KUKA KRL program: MyProgram_135().src

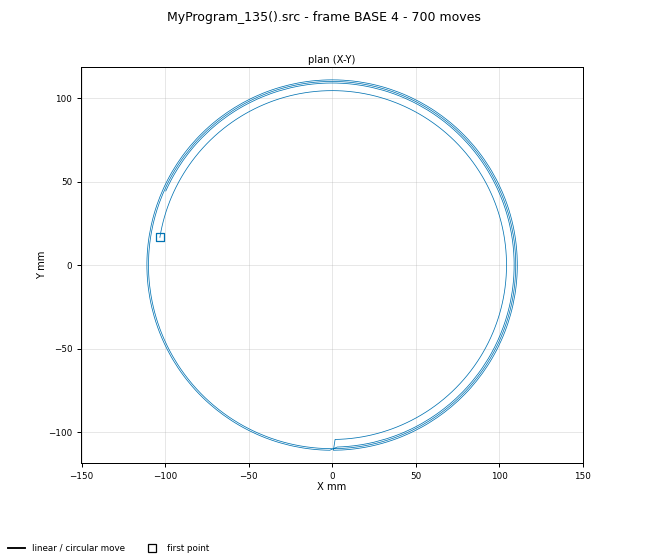
[picture p0: tool path of MyProgram_135().src in frame BASE 4, 700 of 700 moves have a stored position in this frame; points joined in program order, loops and branches not executed]
&ACCESS RVP
&REL 1
&PARAM TEMPLATE = C:\KRC\Roboter\Template\vorgabe
&PARAM EDITMASK = *
DEF MyProgram_135()
; ---- Setting reference (Base) ----
$BASE = BASE_DATA[4]

; --------------------------
; ---- Setting tool (TCP) ----
$TOOL = TOOL_DATA[3]
; --------------------------

$VEL.CP = VEL_APROX_PRINT
Startdeposition()
$VEL.CP = VEL_PRINT
LIN {X -103.1333,Y 16.5825,Z 109,A 165.9038,B 24.9354,C -1.8568,E1 24.8421,E2 279.7377} C_DIS
LIN {X -102.5383,Y 19.9247,Z 109,A 164.1624,B 24.9347,C -1.867,E1 24.843,E2 281.465} C_DIS
LIN {X -101.9199,Y 22.8869,Z 109,A 162.3578,B 24.9347,C -1.8672,E1 24.844,E2 283.2797} C_DIS
LIN {X -101.1577,Y 26.042,Z 109,A 160.77,B 24.9338,C -1.8797,E1 24.8451,E2 284.8471} C_DIS
LIN {X -100.4534,Y 28.6392,Z 109,A 159.199,B 24.9337,C -1.881,E1 24.8463,E2 286.424} C_DIS
LIN {X -99.4092,Y 32.0762,Z 109,A 157.2856,B 24.9331,C -1.8892,E1 24.8479,E2 288.3288} C_DIS
LIN {X -98.5325,Y 34.676,Z 109,A 155.6889,B 24.933,C -1.8907,E1 24.8493,E2 289.9311} C_DIS
LIN {X -97.2525,Y 38.1187,Z 109,A 153.7477,B 24.9324,C -1.8995,E1 24.8512,E2 291.8622} C_DIS
LIN {X -96.2896,Y 40.4893,Z 109,A 152.276,B 24.9322,C -1.9014,E1 24.8528,E2 293.3376} C_DIS
LIN {X -94.9474,Y 43.5478,Z 109,A 150.3049,B 24.9322,C -1.902,E1 24.8551,E2 295.318} C_DIS
LIN {X -93.5406,Y 46.4891,Z 109,A 148.6045,B 24.9316,C -1.9105,E1 24.8571,E2 297.0073} C_DIS
LIN {X -91.8565,Y 49.7339,Z 109,A 146.632,B 24.9311,C -1.9176,E1 24.8597,E2 298.9735} C_DIS
LIN {X -90.2584,Y 52.582,Z 109,A 144.8687,B 24.9306,C -1.9237,E1 24.8621,E2 300.7314} C_DIS
LIN {X -88.786,Y 55.0296,Z 109,A 143.2,B 24.9306,C -1.9246,E1 24.8646,E2 302.4065} C_DIS
LIN {X -87.1648,Y 57.5619,Z 109,A 141.5447,B 24.9302,C -1.9291,E1 24.8671,E2 304.0595} C_DIS
LIN {X -85.388,Y 60.1693,Z 109,A 139.8581,B 24.9298,C -1.9354,E1 24.8698,E2 305.7393} C_DIS
LIN {X -83.8937,Y 62.2359,Z 109,A 138.3455,B 24.9298,C -1.9352,E1 24.8723,E2 307.2598} C_DIS
LIN {X -81.9529,Y 64.7672,Z 109,A 136.6672,B 24.9293,C -1.9424,E1 24.8751,E2 308.9288} C_DIS
LIN {X -79.7445,Y 67.4686,Z 109,A 134.6792,B 24.9291,C -1.9448,E1 24.8787,E2 310.9204} C_DIS
LIN {X -77.5632,Y 69.9655,Z 109,A 132.8296,B 24.9288,C -1.9483,E1 24.8821,E2 312.7698} C_DIS
LIN {X -75.2059,Y 72.4924,Z 109,A 130.9953,B 24.9283,C -1.9552,E1 24.8856,E2 314.5956} C_DIS
LIN {X -72.7466,Y 74.9609,Z 109,A 129.0328,B 24.9281,C -1.9579,E1 24.8895,E2 316.5599} C_DIS
LIN {X -70.3326,Y 77.2305,Z 109,A 127.1463,B 24.928,C -1.9597,E1 24.8934,E2 318.4498} C_DIS
LIN {X -67.7352,Y 79.5174,Z 109,A 125.3395,B 24.9274,C -1.9673,E1 24.8972,E2 320.2456} C_DIS
LIN {X -64.9962,Y 81.7719,Z 109,A 123.3659,B 24.9272,C -1.9706,E1 24.9015,E2 322.2189} C_DIS
LIN {X -62.8029,Y 83.4678,Z 109,A 121.8583,B 24.9269,C -1.9743,E1 24.9048,E2 323.7231} C_DIS
LIN {X -60.123,Y 85.4206,Z 109,A 119.9594,B 24.9269,C -1.975,E1 24.9091,E2 325.6268} C_DIS
LIN {X -57.3874,Y 87.2798,Z 109,A 118.158,B 24.9266,C -1.9791,E1 24.9133,E2 327.4244} C_DIS
LIN {X -54.2739,Y 89.2491,Z 109,A 116.2553,B 24.926,C -1.9872,E1 24.9178,E2 329.314} C_DIS
LIN {X -52.1167,Y 90.5258,Z 109,A 114.8585,B 24.9258,C -1.9889,E1 24.9211,E2 330.7109} C_DIS
LIN {X -49.7124,Y 91.8681,Z 109,A 113.2634,B 24.9258,C -1.9884,E1 24.9251,E2 332.3118} C_DIS
LIN {X -46.4551,Y 93.5574,Z 109,A 111.2906,B 24.9255,C -1.9931,E1 24.93,E2 334.2786} C_DIS
LIN {X -43.4974,Y 94.9708,Z 109,A 109.3318,B 24.9257,C -1.99,E1 24.9349,E2 336.2497} C_DIS
LIN {X -40.495,Y 96.2872,Z 109,A 107.6366,B 24.9253,C -1.9964,E1 24.9393,E2 337.9336} C_DIS
LIN {X -37.0875,Y 97.6504,Z 109,A 105.6975,B 24.9249,C -2.0019,E1 24.9443,E2 339.8639} C_DIS
LIN {X -34.6623,Y 98.5373,Z 109,A 104.2027,B 24.9249,C -2.0008,E1 24.9482,E2 341.3642} C_DIS
LIN {X -31.5292,Y 99.586,Z 109,A 102.2735,B 24.9251,C -1.9986,E1 24.9534,E2 343.3022} C_DIS
LIN {X -28.5461,Y 100.4798,Z 109,A 100.7134,B 24.9246,C -2.006,E1 24.9575,E2 344.8473} C_DIS
LIN {X -25.3785,Y 101.3282,Z 109,A 98.7564,B 24.9249,C -2.0018,E1 24.9628,E2 346.817} C_DIS
LIN {X -22.3293,Y 102.0416,Z 109,A 97.2308,B 24.9242,C -2.0106,E1 24.9669,E2 348.3238} C_DIS
LIN {X -19.631,Y 102.5949,Z 109,A 95.6315,B 24.9244,C -2.0085,E1 24.9713,E2 349.9298} C_DIS
LIN {X -16.2066,Y 103.1915,Z 109,A 93.7524,B 24.9242,C -2.0109,E1 24.9765,E2 351.8049} C_DIS
LIN {X -13.3362,Y 103.6013,Z 109,A 92.1299,B 24.9242,C -2.0107,E1 24.981,E2 353.4292} C_DIS
LIN {X -9.5889,Y 104.015,Z 109,A 90.1169,B 24.924,C -2.0139,E1 24.9866,E2 355.4358} C_DIS
LIN {X -6.3744,Y 104.2632,Z 109,A 88.1851,B 24.9244,C -2.0084,E1 24.992,E2 357.3813} C_DIS
LIN {X -3.091,Y 104.4104,Z 109,A 86.4916,B 24.924,C -2.0132,E1 24.9967,E2 359.0639} C_DIS
LIN {X 0.6428,Y 104.4541,Z 109,A 84.5244,B 24.9237,C -2.0167,E1 25.0022,E2 361.0227} C_DIS
LIN {X 3.337,Y 104.4028,Z 109,A 82.9539,B 24.924,C -2.0133,E1 25.0066,E2 362.6009} C_DIS
LIN {X 6.4284,Y 104.2599,Z 109,A 81.1548,B 24.9243,C -2.0094,E1 25.0116,E2 364.4086} C_DIS
LIN {X 9.683,Y 104.0063,Z 109,A 79.4608,B 24.924,C -2.013,E1 25.0163,E2 366.0931} C_DIS
LIN {X 13.3502,Y 103.5994,Z 109,A 77.4906,B 24.9239,C -2.0147,E1 25.0217,E2 368.0578} C_DIS
LIN {X 16.6067,Y 103.1294,Z 109,A 75.5342,B 24.9244,C -2.0083,E1 25.0272,E2 370.0277} C_DIS
LIN {X 19.6735,Y 102.5867,Z 109,A 73.9793,B 24.924,C -2.0136,E1 25.0314,E2 371.5683} C_DIS
LIN {X 22.8843,Y 101.9205,Z 109,A 72.0241,B 24.9245,C -2.0066,E1 25.0368,E2 373.5375} C_DIS
LIN {X 25.9326,Y 101.1858,Z 109,A 70.5056,B 24.924,C -2.0134,E1 25.0408,E2 375.0374} C_DIS
LIN {X 28.5921,Y 100.4668,Z 109,A 68.9194,B 24.9243,C -2.0095,E1 25.0451,E2 376.6305} C_DIS
LIN {X 32.0776,Y 99.4088,Z 109,A 66.9893,B 24.9243,C -2.0106,E1 25.0503,E2 378.5544} C_DIS
LIN {X 34.6913,Y 98.5271,Z 109,A 65.4074,B 24.9245,C -2.0066,E1 25.0545,E2 380.1427} C_DIS
LIN {X 38.1127,Y 97.2548,Z 109,A 63.4873,B 24.9245,C -2.0079,E1 25.0595,E2 382.0555} C_DIS
LIN {X 40.5037,Y 96.2836,Z 109,A 62.0408,B 24.9246,C -2.0052,E1 25.0632,E2 383.5051} C_DIS
LIN {X 43.5071,Y 94.9663,Z 109,A 60.0932,B 24.9252,C -1.9972,E1 25.0682,E2 385.4667} C_DIS
LIN {X 46.4667,Y 93.5517,Z 109,A 58.4072,B 24.925,C -1.9995,E1 25.0724,E2 387.1429} C_DIS
LIN {X 49.7271,Y 91.8602,Z 109,A 56.4415,B 24.925,C -1.9988,E1 25.0772,E2 389.1048} C_DIS
LIN {X 52.602,Y 90.2469,Z 109,A 54.6726,B 24.9252,C -1.9977,E1 25.0815,E2 390.8709} C_DIS
LIN {X 54.8087,Y 88.9239,Z 109,A 53.0827,B 24.9259,C -1.9884,E1 25.0854,E2 392.4777} C_DIS
LIN {X 57.567,Y 87.1614,Z 109,A 51.3965,B 24.9257,C -1.99,E1 25.0893,E2 394.1548} C_DIS
LIN {X 60.5312,Y 85.1297,Z 109,A 49.4373,B 24.926,C -1.9871,E1 25.0938,E2 396.1139} C_DIS
LIN {X 63.2881,Y 83.1026,Z 109,A 47.5197,B 24.9263,C -1.9821,E1 25.0981,E2 398.0364} C_DIS
LIN {X 65.78,Y 81.1422,Z 109,A 45.8503,B 24.9263,C -1.9818,E1 25.1017,E2 399.7005} C_DIS
LIN {X 68.4304,Y 78.9208,Z 109,A 43.9194,B 24.9267,C -1.9767,E1 25.1058,E2 401.6359} C_DIS
LIN {X 70.8883,Y 76.7206,Z 109,A 42.0884,B 24.9271,C -1.9721,E1 25.1096,E2 403.4702} C_DIS
LIN {X 73.4416,Y 74.2792,Z 109,A 40.2308,B 24.9271,C -1.9713,E1 25.1133,E2 405.322} C_DIS
LIN {X 75.8718,Y 71.7958,Z 109,A 38.2991,B 24.9275,C -1.9661,E1 25.1171,E2 407.2577} C_DIS
LIN {X 78.0198,Y 69.4555,Z 109,A 36.5169,B 24.9279,C -1.9605,E1 25.1204,E2 409.0452} C_DIS
LIN {X 80.342,Y 66.7551,Z 109,A 34.6539,B 24.9279,C -1.9597,E1 25.1238,E2 410.9017} C_DIS
LIN {X 82.571,Y 63.978,Z 109,A 32.7197,B 24.9283,C -1.9557,E1 25.1271,E2 412.8361} C_DIS
LIN {X 84.3727,Y 61.5819,Z 109,A 31.0746,B 24.9286,C -1.9516,E1 25.1299,E2 414.483} C_DIS
LIN {X 86.1363,Y 59.0932,Z 109,A 29.2885,B 24.9292,C -1.9427,E1 25.1327,E2 416.2815} C_DIS
LIN {X 87.944,Y 56.3643,Z 109,A 27.6077,B 24.9292,C -1.9427,E1 25.1353,E2 417.9536} C_DIS
LIN {X 89.8865,Y 53.2117,Z 109,A 25.6766,B 24.9293,C -1.9415,E1 25.1381,E2 419.8778} C_DIS
LIN {X 91.1627,Y 50.9945,Z 109,A 24.2402,B 24.9297,C -1.9364,E1 25.14,E2 421.319} C_DIS
LIN {X 92.7207,Y 48.1077,Z 109,A 22.4502,B 24.93,C -1.9317,E1 25.1424,E2 423.1105} C_DIS
LIN {X 93.9035,Y 45.755,Z 109,A 21.0638,B 24.9302,C -1.9301,E1 25.1441,E2 424.4933} C_DIS
LIN {X 95.2133,Y 42.9593,Z 109,A 19.3763,B 24.9305,C -1.9255,E1 25.1461,E2 426.1824} C_DIS
LIN {X 96.3419,Y 40.3653,Z 109,A 17.779,B 24.931,C -1.9191,E1 25.1478,E2 427.7861} C_DIS
LIN {X 97.6586,Y 37.0659,Z 109,A 15.8954,B 24.9312,C -1.9161,E1 25.1498,E2 429.6664} C_DIS
LIN {X 98.5376,Y 34.6615,Z 109,A 14.4588,B 24.9316,C -1.9106,E1 25.1511,E2 431.108} C_DIS
LIN {X 99.58,Y 31.5485,Z 109,A 12.5172,B 24.9324,C -1.8993,E1 25.1528,E2 433.0654} C_DIS
LIN {X 100.4806,Y 28.5433,Z 109,A 10.9613,B 24.9323,C -1.9009,E1 25.154,E2 434.6083} C_DIS
LIN {X 101.3287,Y 25.3764,Z 109,A 9.0222,B 24.9331,C -1.8895,E1 25.1554,E2 436.5633} C_DIS
LIN {X 102.0383,Y 22.344,Z 109,A 7.4709,B 24.933,C -1.8908,E1 25.1563,E2 438.1026} C_DIS
LIN {X 102.6944,Y 19.1139,Z 109,A 5.5306,B 24.9338,C -1.8795,E1 25.1574,E2 440.0581} C_DIS
LIN {X 103.2485,Y 15.8377,Z 109,A 3.8275,B 24.9338,C -1.8788,E1 25.1581,E2 441.7529} C_DIS
LIN {X 103.7381,Y 12.2265,Z 109,A 1.872,B 24.9341,C -1.8743,E1 25.1588,E2 443.7075} C_DIS
LIN {X 104.0798,Y 8.8756,Z 109,A -0.0838,B 24.9349,C -1.8638,E1 25.1593,E2 445.6765} C_DIS
LIN {X 104.3039,Y 5.6384,Z 109,A -1.761,B 24.9349,C -1.8624,E1 25.1596,E2 447.347} C_DIS
LIN {X 104.4268,Y 2.5486,Z 109,A -3.4231,B 24.9353,C -1.8583,E1 25.1598,E2 449.0088} C_DIS
LIN {X 104.4555,Y -0.4515,Z 109,A -5.045,B 24.9356,C -1.854,E1 25.1598,E2 450.6312} C_DIS
LIN {X 104.4035,Y -3.3159,Z 109,A -6.6414,B 24.936,C -1.8479,E1 25.1597,E2 452.2326} C_DIS
LIN {X 104.2605,Y -6.4198,Z 109,A -8.4376,B 24.9366,C -1.8384,E1 25.1594,E2 454.0404} C_DIS
LIN {X 104.0063,Y -9.6835,Z 109,A -10.1141,B 24.9367,C -1.8376,E1 25.159,E2 455.7088} C_DIS
LIN {X 103.5993,Y -13.351,Z 109,A -12.08,B 24.937,C -1.8335,E1 25.1583,E2 457.6727} C_DIS
LIN {X 103.1318,Y -16.5923,Z 109,A -14.0214,B 24.9378,C -1.8216,E1 25.1575,E2 459.631} C_DIS
LIN {X 102.5862,Y -19.6761,Z 109,A -15.5701,B 24.9377,C -1.8232,E1 25.1567,E2 461.1668} C_DIS
LIN {X 101.9204,Y -22.8849,Z 109,A -17.5078,B 24.9385,C -1.8115,E1 25.1556,E2 463.1208} C_DIS
LIN {X 101.1914,Y -25.9108,Z 109,A -19.0981,B 24.9385,C -1.811,E1 25.1545,E2 464.7031} C_DIS
LIN {X 100.3233,Y -29.0982,Z 109,A -21.0031,B 24.9392,C -1.8013,E1 25.1531,E2 466.6201} C_DIS
LIN {X 99.3755,Y -32.1805,Z 109,A -22.551,B 24.9389,C -1.805,E1 25.1518,E2 468.1504} C_DIS
LIN {X 98.5259,Y -34.6948,Z 109,A -24.0998,B 24.9395,C -1.7965,E1 25.1504,E2 469.7105} C_DIS
LIN {X 97.2495,Y -38.1263,Z 109,A -26.0067,B 24.9396,C -1.7946,E1 25.1485,E2 471.6113} C_DIS
LIN {X 96.289,Y -40.4907,Z 109,A -27.4386,B 24.94,C -1.7889,E1 25.1469,E2 473.0487} C_DIS
LIN {X 94.9752,Y -43.4876,Z 109,A -29.3712,B 24.9408,C -1.7776,E1 25.1447,E2 474.9974} C_DIS
LIN {X 93.5525,Y -46.4651,Z 109,A -31.0647,B 24.9408,C -1.7771,E1 25.1426,E2 476.683} C_DIS
LIN {X 91.8557,Y -49.7354,Z 109,A -33.0409,B 24.9411,C -1.773,E1 25.1401,E2 478.6586} C_DIS
LIN {X 90.2308,Y -52.6292,Z 109,A -34.8042,B 24.9413,C -1.77,E1 25.1376,E2 480.4197} C_DIS
LIN {X 88.9248,Y -54.8074,Z 109,A -36.3703,B 24.942,C -1.7588,E1 25.1353,E2 482.0044} C_DIS
LIN {X 87.1556,Y -57.5759,Z 109,A -38.0575,B 24.942,C -1.7585,E1 25.1328,E2 483.6838} C_DIS
LIN {X 85.1321,Y -60.5279,Z 109,A -39.9916,B 24.9423,C -1.7542,E1 25.1297,E2 485.6185} C_DIS
LIN {X 83.1361,Y -63.2445,Z 109,A -41.9106,B 24.9429,C -1.7462,E1 25.1265,E2 487.5472} C_DIS
LIN {X 81.1408,Y -65.7818,Z 109,A -43.5911,B 24.9429,C -1.7453,E1 25.1235,E2 489.2221} C_DIS
LIN {X 78.9092,Y -68.4436,Z 109,A -45.5258,B 24.9433,C -1.7391,E1 25.12,E2 491.1627} C_DIS
LIN {X 76.7241,Y -70.8844,Z 109,A -47.3968,B 24.9438,C -1.7314,E1 25.1165,E2 493.0434} C_DIS
LIN {X 74.2989,Y -73.4217,Z 109,A -49.1872,B 24.9438,C -1.7322,E1 25.113,E2 494.8242} C_DIS
LIN {X 71.8174,Y -75.8516,Z 109,A -51.1224,B 24.9441,C -1.7264,E1 25.1091,E2 496.7652} C_DIS
LIN {X 69.465,Y -78.0113,Z 109,A -52.9083,B 24.9445,C -1.7209,E1 25.1054,E2 498.5569} C_DIS
LIN {X 66.7697,Y -80.3298,Z 109,A -54.7742,B 24.9445,C -1.7199,E1 25.1014,E2 500.4178} C_DIS
LIN {X 63.972,Y -82.5755,Z 109,A -56.7153,B 24.9448,C -1.7167,E1 25.0972,E2 502.3592} C_DIS
LIN {X 61.7725,Y -84.2332,Z 109,A -58.2229,B 24.945,C -1.7137,E1 25.0938,E2 503.8686} C_DIS
LIN {X 59.0546,Y -86.1625,Z 109,A -60.1621,B 24.9455,C -1.7053,E1 25.0893,E2 505.8209} C_DIS
LIN {X 56.3488,Y -87.9539,Z 109,A -61.8347,B 24.9455,C -1.7063,E1 25.0854,E2 507.4858} C_DIS
LIN {X 53.2184,Y -89.8826,Z 109,A -63.7615,B 24.9455,C -1.7062,E1 25.0809,E2 509.4068} C_DIS
LIN {X 50.6913,Y -91.332,Z 109,A -65.5093,B 24.946,C -1.6972,E1 25.0766,E2 511.1707} C_DIS
LIN {X 47.564,Y -92.9986,Z 109,A -67.2876,B 24.9458,C -1.7006,E1 25.0722,E2 512.9359} C_DIS
LIN {X 44.9999,Y -94.2664,Z 109,A -68.905,B 24.9461,C -1.6961,E1 25.0681,E2 514.5597} C_DIS
LIN {X 41.8121,Y -95.7227,Z 109,A -70.8092,B 24.9462,C -1.6939,E1 25.0633,E2 516.4644} C_DIS
LIN {X 38.7975,Y -96.9857,Z 109,A -72.7555,B 24.9468,C -1.6851,E1 25.0582,E2 518.4271} C_DIS
LIN {X 35.8621,Y -98.107,Z 109,A -74.2753,B 24.9464,C -1.691,E1 25.0543,E2 519.9296} C_DIS
LIN {X 33.2923,Y -99.0086,Z 109,A -75.8498,B 24.9467,C -1.6858,E1 25.0501,E2 521.5133} C_DIS
LIN {X 29.7546,Y -100.1286,Z 109,A -77.7944,B 24.9467,C -1.6871,E1 25.0449,E2 523.4513} C_DIS
LIN {X 27.1413,Y -100.8684,Z 109,A -79.368,B 24.947,C -1.6821,E1 25.0407,E2 525.0342} C_DIS
LIN {X 23.5848,Y -101.7587,Z 109,A -81.2877,B 24.9469,C -1.6838,E1 25.0355,E2 526.9472} C_DIS
LIN {X 21.0894,Y -102.305,Z 109,A -82.7339,B 24.9471,C -1.6807,E1 25.0315,E2 528.3988} C_DIS
LIN {X 17.8473,Y -102.922,Z 109,A -84.6152,B 24.9473,C -1.6764,E1 25.0263,E2 530.2882} C_DIS
LIN {X 14.7433,Y -103.4104,Z 109,A -86.2534,B 24.9472,C -1.6786,E1 25.0218,E2 531.9196} C_DIS
LIN {X 11.5014,Y -103.8228,Z 109,A -88.1968,B 24.9476,C -1.6715,E1 25.0164,E2 533.8784} C_DIS
LIN {X 8.2018,Y -104.1336,Z 109,A -89.9621,B 24.9476,C -1.6727,E1 25.0115,E2 535.64} C_DIS
LIN {X 4.4645,Y -104.3606,Z 109,A -91.8665,B 24.9473,C -1.6777,E1 25.0062,E2 537.5317} C_DIS
LIN {X 1.7914,Y -104.4408,Z 109,A -93.4225,B 24.9475,C -1.6738,E1 25.0018,E2 539.0968} C_DIS
LIN {X 1.7914,Y -104.4408,Z 109,A -93.4225,B 24.9475,C -1.6738,E1 25.0018,E2 539.0968} C_DIS
Enddeposition()
LIN {X 0.7724,Y -110.9124,Z 110,A -93.2398,B 24.9521,C -1.5986,E1 25.0018,E2 539.0923} C_DIS
Startdeposition()
$VEL.CP = VEL_PRINT
LIN {X 3.161,Y -110.8717,Z 110,A -91.8429,B 24.9517,C -1.6059,E1 25.0058,E2 537.6783} C_DIS
LIN {X 5.7879,Y -110.7659,Z 110,A -90.625,B 24.952,C -1.6004,E1 25.0091,E2 536.4738} C_DIS
LIN {X 8.5045,Y -110.5905,Z 110,A -89.058,B 24.9516,C -1.6079,E1 25.0136,E2 534.8897} C_DIS
LIN {X 11.216,Y -110.3485,Z 110,A -87.8156,B 24.9519,C -1.6017,E1 25.017,E2 533.6629} C_DIS
LIN {X 13.9207,Y -110.04,Z 110,A -86.411,B 24.9519,C -1.6025,E1 25.0209,E2 532.2575} C_DIS
LIN {X 16.617,Y -109.6652,Z 110,A -84.8446,B 24.9514,C -1.6103,E1 25.0252,E2 530.6739} C_DIS
LIN {X 18.9628,Y -109.2856,Z 110,A -83.4902,B 24.951,C -1.6167,E1 25.029,E2 529.3057} C_DIS
LIN {X 21.6391,Y -108.7873,Z 110,A -82.0759,B 24.951,C -1.6183,E1 25.0329,E2 527.8895} C_DIS
LIN {X 24.3024,Y -108.2235,Z 110,A -80.8122,B 24.9512,C -1.6134,E1 25.0363,E2 526.639} C_DIS
LIN {X 26.951,Y -107.5945,Z 110,A -79.2797,B 24.9508,C -1.6203,E1 25.0405,E2 525.0924} C_DIS
LIN {X 30.0786,Y -106.7604,Z 110,A -77.7027,B 24.9509,C -1.618,E1 25.0447,E2 523.5234} C_DIS
LIN {X 33.0142,Y -105.8894,Z 110,A -76.0985,B 24.9508,C -1.6208,E1 25.049,E2 521.9154} C_DIS
LIN {X 36.4094,Y -104.7709,Z 110,A -74.483,B 24.9512,C -1.613,E1 25.0532,E2 520.3214} C_DIS
LIN {X 38.9696,Y -103.8458,Z 110,A -72.9425,B 24.9508,C -1.6208,E1 25.0573,E2 518.7659} C_DIS
LIN {X 41.5064,Y -102.8581,Z 110,A -71.6788,B 24.951,C -1.6165,E1 25.0606,E2 517.515} C_DIS
LIN {X 44.1998,Y -101.7294,Z 110,A -70.2679,B 24.9512,C -1.6145,E1 25.0642,E2 516.1122} C_DIS
LIN {X 46.1898,Y -100.8436,Z 110,A -68.8916,B 24.9504,C -1.6272,E1 25.0677,E2 514.7093} C_DIS
LIN {X 48.9607,Y -99.526,Z 110,A -67.3122,B 24.9502,C -1.6295,E1 25.0717,E2 513.1285} C_DIS
LIN {X 51.3884,Y -98.2945,Z 110,A -65.911,B 24.9502,C -1.6317,E1 25.0752,E2 511.7261} C_DIS
LIN {X 53.4831,Y -97.1724,Z 110,A -64.5863,B 24.9497,C -1.6381,E1 25.0785,E2 510.39} C_DIS
LIN {X 55.8518,Y -95.8306,Z 110,A -63.2874,B 24.9499,C -1.6359,E1 25.0816,E2 509.1002} C_DIS
LIN {X 58.1867,Y -94.4311,Z 110,A -61.7578,B 24.9494,C -1.644,E1 25.0853,E2 507.5562} C_DIS
LIN {X 60.7755,Y -92.7843,Z 110,A -60.4702,B 24.95,C -1.634,E1 25.0882,E2 506.2967} C_DIS
LIN {X 62.7502,Y -91.4623,Z 110,A -58.9573,B 24.949,C -1.6491,E1 25.0918,E2 504.7531} C_DIS
LIN {X 65.255,Y -89.6904,Z 110,A -57.6703,B 24.9497,C -1.6392,E1 25.0947,E2 503.494} C_DIS
LIN {X 67.1624,Y -88.2731,Z 110,A -56.1577,B 24.9487,C -1.6544,E1 25.0981,E2 501.9508} C_DIS
LIN {X 69.5773,Y -86.3804,Z 110,A -54.8707,B 24.9493,C -1.6447,E1 25.1009,E2 500.6917} C_DIS
LIN {X 71.4129,Y -84.8713,Z 110,A -53.3586,B 24.9484,C -1.6601,E1 25.1042,E2 499.1489} C_DIS
LIN {X 73.732,Y -82.8624,Z 110,A -51.9104,B 24.9485,C -1.6577,E1 25.1072,E2 497.7122} C_DIS
LIN {X 75.4913,Y -81.265,Z 110,A -50.5603,B 24.948,C -1.6661,E1 25.11,E2 496.3478} C_DIS
LIN {X 77.709,Y -79.1447,Z 110,A -49.2734,B 24.9486,C -1.6566,E1 25.1125,E2 495.0887} C_DIS
LIN {X 79.3878,Y -77.4629,Z 110,A -47.7092,B 24.9474,C -1.6747,E1 25.1156,E2 493.4884} C_DIS
LIN {X 81.265,Y -75.4913,Z 110,A -46.4925,B 24.9478,C -1.6697,E1 25.1179,E2 492.2888} C_DIS
LIN {X 83.0931,Y -73.4742,Z 110,A -44.9652,B 24.9472,C -1.6788,E1 25.1208,E2 490.7469} C_DIS
LIN {X 85.0924,Y -71.1468,Z 110,A -43.6794,B 24.9478,C -1.6695,E1 25.1231,E2 489.4889} C_DIS
LIN {X 86.5983,Y -69.3085,Z 110,A -42.1687,B 24.9468,C -1.6855,E1 25.1258,E2 487.9474} C_DIS
LIN {X 88.4809,Y -66.8858,Z 110,A -40.8831,B 24.9473,C -1.6763,E1 25.1279,E2 486.6895} C_DIS
LIN {X 89.8948,Y -64.9759,Z 110,A -39.3728,B 24.9463,C -1.6924,E1 25.1305,E2 485.1484} C_DIS
LIN {X 91.6562,Y -62.4637,Z 110,A -37.9332,B 24.9465,C -1.6903,E1 25.1327,E2 483.7209} C_DIS
LIN {X 92.9747,Y -60.4867,Z 110,A -36.5771,B 24.9459,C -1.6996,E1 25.1348,E2 482.3497} C_DIS
LIN {X 94.6108,Y -57.8911,Z 110,A -35.1309,B 24.9459,C -1.6979,E1 25.1369,E2 480.9148} C_DIS
LIN {X 96.003,Y -55.5518,Z 110,A -33.6701,B 24.9456,C -1.7045,E1 25.139,E2 479.4461} C_DIS
LIN {X 97.8214,Y -52.2867,Z 110,A -31.8148,B 24.9454,C -1.7067,E1 25.1415,E2 477.5951} C_DIS
LIN {X 99.0752,Y -49.8702,Z 110,A -30.2888,B 24.9448,C -1.7164,E1 25.1434,E2 476.0546} C_DIS
LIN {X 100.4152,Y -47.1102,Z 110,A -28.8429,B 24.9448,C -1.7149,E1 25.1452,E2 474.6199} C_DIS
LIN {X 101.4028,Y -44.9488,Z 110,A -27.4947,B 24.9443,C -1.7241,E1 25.1467,E2 473.2573} C_DIS
LIN {X 102.4754,Y -42.4467,Z 110,A -26.0638,B 24.9439,C -1.7296,E1 25.1483,E2 471.8214} C_DIS
LIN {X 103.4862,Y -39.919,Z 110,A -24.7009,B 24.9438,C -1.7319,E1 25.1496,E2 470.4605} C_DIS
LIN {X 104.4347,Y -37.3673,Z 110,A -23.4326,B 24.9439,C -1.7301,E1 25.1508,E2 469.2038} C_DIS
LIN {X 105.3368,Y -34.742,Z 110,A -22.0333,B 24.9437,C -1.733,E1 25.1521,E2 467.8054} C_DIS
LIN {X 106.2409,Y -31.8663,Z 110,A -20.623,B 24.9438,C -1.7313,E1 25.1532,E2 466.4072} C_DIS
LIN {X 106.9007,Y -29.5834,Z 110,A -19.1137,B 24.9427,C -1.748,E1 25.1544,E2 464.8672} C_DIS
LIN {X 107.6765,Y -26.6149,Z 110,A -17.6682,B 24.9428,C -1.7467,E1 25.1554,E2 463.433} C_DIS
LIN {X 108.3266,Y -23.8299,Z 110,A -16.2471,B 24.9427,C -1.7489,E1 25.1563,E2 462.015} C_DIS
LIN {X 109.1059,Y -19.962,Z 110,A -14.3381,B 24.9427,C -1.7496,E1 25.1573,E2 460.1155} C_DIS
LIN {X 109.5101,Y -17.6203,Z 110,A -12.8291,B 24.9415,C -1.7664,E1 25.158,E2 458.5758} C_DIS
LIN {X 109.9095,Y -14.9275,Z 110,A -11.4329,B 24.9413,C -1.7705,E1 25.1585,E2 457.1781} C_DIS
LIN {X 110.2427,Y -12.2257,Z 110,A -10.165,B 24.9413,C -1.7687,E1 25.1589,E2 455.9218} C_DIS
LIN {X 110.5096,Y -9.5165,Z 110,A -8.6398,B 24.9407,C -1.7787,E1 25.1593,E2 454.3821} C_DIS
LIN {X 110.7098,Y -6.8016,Z 110,A -7.2433,B 24.9404,C -1.7829,E1 25.1596,E2 452.9842} C_DIS
LIN {X 110.8434,Y -4.0826,Z 110,A -5.8469,B 24.9401,C -1.787,E1 25.1597,E2 451.5864} C_DIS
LIN {X 110.9102,Y -1.3611,Z 110,A -4.5408,B 24.9401,C -1.787,E1 25.1597,E2 450.288} C_DIS
LIN {X 110.8986,Y 1.9937,Z 110,A -2.9486,B 24.9401,C -1.7862,E1 25.1597,E2 448.7071} C_DIS
LIN {X 110.7659,Y 5.7879,Z 110,A -1.0715,B 24.9401,C -1.7887,E1 25.1595,E2 446.8352} C_DIS
LIN {X 110.5905,Y 8.5045,Z 110,A 0.5294,B 24.9391,C -1.8021,E1 25.1592,E2 445.2123} C_DIS
LIN {X 110.2427,Y 12.2257,Z 110,A 2.4036,B 24.9389,C -1.8057,E1 25.1587,E2 443.3407} C_DIS
LIN {X 109.9095,Y 14.9275,Z 110,A 3.9291,B 24.9382,C -1.8156,E1 25.1581,E2 441.8009} C_DIS
LIN {X 109.453,Y 17.9615,Z 110,A 5.2493,B 24.9387,C -1.8087,E1 25.1576,E2 440.5048} C_DIS
LIN {X 108.9793,Y 20.6422,Z 110,A 6.6101,B 24.9385,C -1.811,E1 25.1569,E2 439.1464} C_DIS
LIN {X 108.4398,Y 23.3105,Z 110,A 8.2506,B 24.9375,C -1.826,E1 25.156,E2 437.4801} C_DIS
LIN {X 107.5945,Y 26.951,Z 110,A 10.2146,B 24.937,C -1.8335,E1 25.1547,E2 435.5097} C_DIS
LIN {X 106.8064,Y 29.9163,Z 110,A 11.4991,B 24.9376,C -1.8248,E1 25.1537,E2 434.2532} C_DIS
LIN {X 105.7393,Y 33.4981,Z 110,A 13.7072,B 24.9363,C -1.8432,E1 25.1519,E2 432.0143} C_DIS
LIN {X 104.7709,Y 36.4094,Z 110,A 15.1531,B 24.9364,C -1.8417,E1 25.1506,E2 430.5801} C_DIS
LIN {X 103.8458,Y 38.9696,Z 110,A 16.3891,B 24.9367,C -1.8382,E1 25.1495,E2 429.3591} C_DIS
LIN {X 102.8581,Y 41.5064,Z 110,A 17.7866,B 24.9364,C -1.842,E1 25.148,E2 427.9606} C_DIS
LIN {X 101.8085,Y 44.0182,Z 110,A 19.3455,B 24.9356,C -1.8529,E1 25.1463,E2 426.3844} C_DIS
LIN {X 100.6976,Y 46.5034,Z 110,A 20.7431,B 24.9354,C -1.8566,E1 25.1447,E2 424.9858} C_DIS
LIN {X 99.6797,Y 48.6507,Z 110,A 21.9632,B 24.9352,C -1.8597,E1 25.1432,E2 423.765} C_DIS
LIN {X 98.2945,Y 51.3884,Z 110,A 23.5386,B 24.9349,C -1.8637,E1 25.1412,E2 422.1884} C_DIS
LIN {X 96.9134,Y 53.9471,Z 110,A 24.9708,B 24.9349,C -1.8647,E1 25.1393,E2 420.7613} C_DIS
LIN {X 95.6546,Y 56.1496,Z 110,A 26.1732,B 24.9349,C -1.8634,E1 25.1376,E2 419.5682} C_DIS
LIN {X 94.4311,Y 58.1867,Z 110,A 27.6841,B 24.9338,C -1.8793,E1 25.1354,E2 418.0274} C_DIS
LIN {X 92.6306,Y 61.0085,Z 110,A 29.2114,B 24.9341,C -1.8749,E1 25.1331,E2 416.5183} C_DIS
LIN {X 91.2648,Y 63.0342,Z 110,A 30.3682,B 24.9342,C -1.8734,E1 25.1313,E2 415.3707} C_DIS
LIN {X 89.6904,Y 65.255,Z 110,A 31.968,B 24.9334,C -1.8855,E1 25.1286,E2 413.7499} C_DIS
LIN {X 88.0619,Y 67.4365,Z 110,A 33.3273,B 24.9333,C -1.8869,E1 25.1264,E2 412.3938} C_DIS
LIN {X 86.3804,Y 69.5773,Z 110,A 34.7264,B 24.933,C -1.89,E1 25.1239,E2 410.994} C_DIS
LIN {X 84.6469,Y 71.6762,Z 110,A 36.167,B 24.9327,C -1.8948,E1 25.1213,E2 409.5486} C_DIS
LIN {X 82.8624,Y 73.732,Z 110,A 37.5246,B 24.9327,C -1.8959,E1 25.1188,E2 408.1946} C_DIS
LIN {X 81.265,Y 75.4913,Z 110,A 38.8752,B 24.932,C -1.9041,E1 25.1163,E2 406.8306} C_DIS
LIN {X 79.1447,Y 77.709,Z 110,A 40.4124,B 24.932,C -1.9055,E1 25.1133,E2 405.2968} C_DIS
LIN {X 76.4829,Y 80.3325,Z 110,A 42.2458,B 24.932,C -1.9052,E1 25.1096,E2 403.4716} C_DIS
LIN {X 74.2306,Y 82.416,Z 110,A 43.6619,B 24.9322,C -1.9011,E1 25.1067,E2 402.071} C_DIS
LIN {X 72.1857,Y 84.2129,Z 110,A 45.2241,B 24.9316,C -1.9107,E1 25.1034,E2 400.4923} C_DIS
LIN {X 70.0972,Y 85.959,Z 110,A 46.4627,B 24.9319,C -1.906,E1 25.1008,E2 399.2694} C_DIS
LIN {X 67.9408,Y 87.6733,Z 110,A 48.0306,B 24.9313,C -1.915,E1 25.0973,E2 397.6861} C_DIS
LIN {X 65.795,Y 89.295,Z 110,A 49.2642,B 24.9316,C -1.9107,E1 25.0946,E2 396.4672} C_DIS
LIN {X 63.5838,Y 90.8828,Z 110,A 50.8273,B 24.9309,C -1.9199,E1 25.091,E2 394.8877} C_DIS
LIN {X 61.6231,Y 92.2254,Z 110,A 52.0504,B 24.9308,C -1.9217,E1 25.0881,E2 393.6645} C_DIS
LIN {X 59.3412,Y 93.71,Z 110,A 53.5811,B 24.9302,C -1.9293,E1 25.0845,E2 392.1207} C_DIS
LIN {X 57.0235,Y 95.138,Z 110,A 54.8536,B 24.9305,C -1.9257,E1 25.0815,E2 390.8609} C_DIS
LIN {X 54.3695,Y 96.6775,Z 110,A 56.2716,B 24.9308,C -1.9208,E1 25.0781,E2 389.4587} C_DIS
LIN {X 52.2867,Y 97.8214,Z 110,A 57.7869,B 24.9298,C -1.9348,E1 25.0743,E2 387.9145} C_DIS
LIN {X 49.5603,Y 99.2288,Z 110,A 59.2381,B 24.9301,C -1.9311,E1 25.0707,E2 386.476} C_DIS
LIN {X 47.4238,Y 100.2692,Z 110,A 60.4624,B 24.93,C -1.9325,E1 25.0676,E2 385.2517} C_DIS
LIN {X 44.9488,Y 101.4028,Z 110,A 61.9945,B 24.9295,C -1.9395,E1 25.0637,E2 383.7068} C_DIS
LIN {X 42.4467,Y 102.4754,Z 110,A 63.3976,B 24.9294,C -1.9408,E1 25.0601,E2 382.3038} C_DIS
LIN {X 39.919,Y 103.4862,Z 110,A 64.8385,B 24.9292,C -1.9437,E1 25.0563,E2 380.8592} C_DIS
LIN {X 37.3407,Y 104.4441,Z 110,A 66.2078,B 24.9292,C -1.9428,E1 25.0528,E2 379.4949} C_DIS
LIN {X 34.7931,Y 105.3203,Z 110,A 67.5617,B 24.9292,C -1.9424,E1 25.0492,E2 378.1447} C_DIS
LIN {X 32.198,Y 106.1425,Z 110,A 68.8824,B 24.9295,C -1.9398,E1 25.0457,E2 376.8324} C_DIS
LIN {X 29.5834,Y 106.9007,Z 110,A 70.4162,B 24.929,C -1.9462,E1 25.0415,E2 375.2861} C_DIS
LIN {X 26.951,Y 107.5945,Z 110,A 71.8207,B 24.929,C -1.947,E1 25.0377,E2 373.8818} C_DIS
LIN {X 24.3024,Y 108.2235,Z 110,A 73.2251,B 24.9289,C -1.9476,E1 25.0339,E2 372.4778} C_DIS
LIN {X 21.2593,Y 108.8604,Z 110,A 74.6859,B 24.9293,C -1.9423,E1 25.0299,E2 371.0315} C_DIS
LIN {X 18.6216,Y 109.3426,Z 110,A 76.1033,B 24.9291,C -1.9441,E1 25.026,E2 369.6112} C_DIS
LIN {X 15.9326,Y 109.7667,Z 110,A 77.5388,B 24.9291,C -1.9458,E1 25.0221,E2 368.1732} C_DIS
LIN {X 12.2257,Y 110.2427,Z 110,A 79.5489,B 24.9288,C -1.9494,E1 25.0165,E2 366.1558} C_DIS
LIN {X 9.1717,Y 110.5371,Z 110,A 81.004,B 24.9291,C -1.9442,E1 25.0125,E2 364.714} C_DIS
LIN {X 6.8016,Y 110.7098,Z 110,A 82.3612,B 24.9287,C -1.9496,E1 25.0086,E2 363.3446} C_DIS
LIN {X 3.4495,Y 110.8628,Z 110,A 83.8736,B 24.9294,C -1.9403,E1 25.0045,E2 361.8547} C_DIS
LIN {X -0.346,Y 110.9165,Z 110,A 85.7639,B 24.9297,C -1.937,E1 24.9992,E2 359.9722} C_DIS
LIN {X -3.0679,Y 110.8746,Z 110,A 87.1765,B 24.9297,C -1.937,E1 24.9953,E2 358.5597} C_DIS
LIN {X -5.7879,Y 110.7659,Z 110,A 88.5785,B 24.9297,C -1.9363,E1 24.9914,E2 357.159} C_DIS
LIN {X -9.5165,Y 110.5096,Z 110,A 90.8037,B 24.9289,C -1.9475,E1 24.9851,E2 354.9062} C_DIS
LIN {X -12.2257,Y 110.2427,Z 110,A 92.2114,B 24.9289,C -1.9468,E1 24.9812,E2 353.4993} C_DIS
LIN {X -14.9275,Y 109.9095,Z 110,A 93.6195,B 24.9289,C -1.946,E1 24.9773,E2 352.0921} C_DIS
LIN {X -17.9615,Y 109.453,Z 110,A 94.914,B 24.9299,C -1.9331,E1 24.9738,E2 350.8271} C_DIS
LIN {X -20.6422,Y 108.9793,Z 110,A 96.3228,B 24.93,C -1.9321,E1 24.9699,E2 349.4192} C_DIS
LIN {X -23.3105,Y 108.4398,Z 110,A 97.7319,B 24.93,C -1.931,E1 24.9661,E2 348.0111} C_DIS
LIN {X -25.8522,Y 107.8626,Z 110,A 99.1351,B 24.93,C -1.9321,E1 24.9623,E2 346.6035} C_DIS
LIN {X -28.6033,Y 107.1654,Z 110,A 100.713,B 24.9298,C -1.9352,E1 24.958,E2 345.016} C_DIS
LIN {X -31.0852,Y 106.4726,Z 110,A 102.1,B 24.9298,C -1.936,E1 24.9542,E2 343.6247} C_DIS
LIN {X -33.8272,Y 105.6328,Z 110,A 103.5324,B 24.93,C -1.9323,E1 24.9504,E2 342.1986} C_DIS
LIN {X -36.4094,Y 104.7709,Z 110,A 104.9422,B 24.9301,C -1.9307,E1 24.9467,E2 340.7898} C_DIS
LIN {X -38.9696,Y 103.8458,Z 110,A 106.1896,B 24.9307,C -1.9225,E1 24.9435,E2 339.5595} C_DIS
LIN {X -41.5064,Y 102.8581,Z 110,A 107.5997,B 24.9308,C -1.9207,E1 24.9398,E2 338.1505} C_DIS
LIN {X -44.0182,Y 101.8085,Z 110,A 109.0104,B 24.931,C -1.9189,E1 24.9362,E2 336.741} C_DIS
LIN {X -46.1898,Y 100.8436,Z 110,A 110.4052,B 24.9306,C -1.9237,E1 24.9326,E2 335.3314} C_DIS
LIN {X -48.6507,Y 99.6797,Z 110,A 111.8161,B 24.9308,C -1.9217,E1 24.9291,E2 333.9217} C_DIS
LIN {X -51.3884,Y 98.2945,Z 110,A 113.4069,B 24.9309,C -1.9193,E1 24.9251,E2 332.3322} C_DIS
LIN {X -53.4831,Y 97.1724,Z 110,A 114.6389,B 24.9311,C -1.9173,E1 24.9221,E2 331.1013} C_DIS
LIN {X -56.2934,Y 95.5696,Z 110,A 116.0743,B 24.932,C -1.905,E1 24.9187,E2 329.6909} C_DIS
LIN {X -58.4802,Y 94.2478,Z 110,A 117.642,B 24.9314,C -1.9124,E1 24.9149,E2 328.1009} C_DIS
LIN {X -60.7755,Y 92.7843,Z 110,A 118.8907,B 24.9321,C -1.9035,E1 24.912,E2 326.8694} C_DIS
LIN {X -62.7502,Y 91.4623,Z 110,A 120.4494,B 24.9313,C -1.9141,E1 24.9083,E2 325.2802} C_DIS
LIN {X -65.3276,Y 89.6372,Z 110,A 121.8942,B 24.9321,C -1.9034,E1 24.9051,E2 323.8558} C_DIS
LIN {X -67.1624,Y 88.2731,Z 110,A 123.2423,B 24.9318,C -1.9075,E1 24.9021,E2 322.4932} C_DIS
LIN {X -69.3085,Y 86.5983,Z 110,A 124.5248,B 24.9324,C -1.8995,E1 24.8993,E2 321.2247} C_DIS
LIN {X -71.4129,Y 84.8713,Z 110,A 126.0682,B 24.9322,C -1.9018,E1 24.896,E2 319.67} C_DIS
LIN {X -73.4742,Y 83.0931,Z 110,A 127.4855,B 24.9324,C -1.899,E1 24.893,E2 318.2538} C_DIS
LIN {X -75.7475,Y 81.0241,Z 110,A 128.945,B 24.933,C -1.8903,E1 24.89,E2 316.8092} C_DIS
LIN {X -77.709,Y 79.1447,Z 110,A 130.1945,B 24.9337,C -1.8809,E1 24.8875,E2 315.5768} C_DIS
LIN {X -79.3878,Y 77.4629,Z 110,A 131.7221,B 24.9331,C -1.8896,E1 24.8845,E2 314.0219} C_DIS
LIN {X -81.265,Y 75.4913,Z 110,A 133.0056,B 24.9337,C -1.8813,E1 24.8821,E2 312.7526} C_DIS
LIN {X -83.3207,Y 73.2136,Z 110,A 134.4358,B 24.9344,C -1.8713,E1 24.8794,E2 311.34} C_DIS
LIN {X -84.8713,Y 71.4129,Z 110,A 135.8339,B 24.9341,C -1.8747,E1 24.8769,E2 309.9273} C_DIS
LIN {X -86.5983,Y 69.3085,Z 110,A 137.2482,B 24.9344,C -1.8713,E1 24.8744,E2 308.5145} C_DIS
LIN {X -88.2731,Y 67.1624,Z 110,A 138.6627,B 24.9346,C -1.8679,E1 24.872,E2 307.1015} C_DIS
LIN {X -89.8948,Y 64.9759,Z 110,A 140.2076,B 24.9345,C -1.8694,E1 24.8694,E2 305.5454} C_DIS
LIN {X -91.6562,Y 62.4637,Z 110,A 141.6716,B 24.9351,C -1.8603,E1 24.8671,E2 304.0958} C_DIS
LIN {X -92.9747,Y 60.4867,Z 110,A 143.0372,B 24.935,C -1.8622,E1 24.865,E2 302.7189} C_DIS
LIN {X -94.6108,Y 57.8911,Z 110,A 144.4119,B 24.9359,C -1.8496,E1 24.863,E2 301.3673} C_DIS
LIN {X -95.8306,Y 55.8518,Z 110,A 145.7368,B 24.9359,C -1.8498,E1 24.8611,E2 300.0351} C_DIS
LIN {X -97.1724,Y 53.4831,Z 110,A 147.152,B 24.9361,C -1.846,E1 24.8592,E2 298.6214} C_DIS
LIN {X -98.4557,Y 51.0823,Z 110,A 148.6791,B 24.9361,C -1.8465,E1 24.8572,E2 297.0851} C_DIS
LIN {X -99.8295,Y 48.3389,Z 110,A 149.9987,B 24.9371,C -1.8315,E1 24.8556,E2 295.794} C_DIS
LIN {X -100.9858,Y 45.8744,Z 110,A 151.578,B 24.937,C -1.834,E1 24.8538,E2 294.2002} C_DIS
LIN {X -102.0843,Y 43.3748,Z 110,A 152.8302,B 24.9377,C -1.8236,E1 24.8524,E2 292.966} C_DIS
LIN {X -103.0961,Y 40.9122,Z 110,A 154.243,B 24.9379,C -1.8208,E1 24.8509,E2 291.5519} C_DIS
LIN {X -104.0869,Y 38.3211,Z 110,A 155.825,B 24.9378,C -1.8221,E1 24.8493,E2 289.958} C_DIS
LIN {X -104.8854,Y 36.083,Z 110,A 157.1914,B 24.9377,C -1.8235,E1 24.8481,E2 288.5802} C_DIS
LIN {X -105.7394,Y 33.4981,Z 110,A 158.6074,B 24.9379,C -1.8195,E1 24.8469,E2 287.1658} C_DIS
LIN {X -106.5296,Y 30.893,Z 110,A 160.0232,B 24.9382,C -1.8154,E1 24.8458,E2 285.7515} C_DIS
LIN {X -107.347,Y 27.914,Z 110,A 161.5511,B 24.9387,C -1.8077,E1 24.8447,E2 284.233} C_DIS
LIN {X -108.3329,Y 23.8007,Z 110,A 163.6434,B 24.9395,C -1.7972,E1 24.8434,E2 282.1536} C_DIS
LIN {X -109.1059,Y 19.962,Z 110,A 165.5729,B 24.9401,C -1.7871,E1 24.8423,E2 280.2367} C_DIS
LIN {X -109.5101,Y 17.6203,Z 110,A 167.1036,B 24.9396,C -1.7948,E1 24.8416,E2 278.6787} C_DIS
LIN {X -109.9095,Y 14.9275,Z 110,A 168.5195,B 24.9399,C -1.7906,E1 24.8411,E2 277.2644} C_DIS
LIN {X -110.2427,Y 12.2257,Z 110,A 169.805,B 24.9405,C -1.7814,E1 24.8407,E2 275.9931} C_DIS
LIN {X -110.5096,Y 9.5165,Z 110,A 171.3519,B 24.9405,C -1.7822,E1 24.8403,E2 274.4348} C_DIS
LIN {X -110.7098,Y 6.8016,Z 110,A 172.7681,B 24.9407,C -1.778,E1 24.84,E2 273.0202} C_DIS
LIN {X -110.8434,Y 4.0826,Z 110,A 174.1842,B 24.941,C -1.7739,E1 24.8399,E2 271.6055} C_DIS
LIN {X -110.9102,Y 1.3611,Z 110,A 175.5537,B 24.9414,C -1.7679,E1 24.8398,E2 270.242} C_DIS
LIN {X -110.8995,Y -1.9461,Z 110,A 177.112,B 24.9422,C -1.7566,E1 24.8398,E2 268.7012} C_DIS
LIN {X -110.7659,Y -5.7879,Z 110,A 179.0264,B 24.9428,C -1.7475,E1 24.84,E2 266.7971} C_DIS
LIN {X -110.5905,Y -8.5045,Z 110,A -179.3691,B 24.9426,C -1.7506,E1 24.8403,E2 265.1756} C_DIS
LIN {X -110.3485,Y -11.216,Z 110,A -178.1416,B 24.9433,C -1.7392,E1 24.8407,E2 263.9678} C_DIS
LIN {X -110.04,Y -13.9207,Z 110,A -176.7254,B 24.9436,C -1.7351,E1 24.8411,E2 262.553} C_DIS
LIN {X -109.6652,Y -16.617,Z 110,A -175.1457,B 24.9434,C -1.7373,E1 24.8418,E2 260.9585} C_DIS
LIN {X -109.2856,Y -18.9628,Z 110,A -173.7795,B 24.9434,C -1.7387,E1 24.8424,E2 259.5807} C_DIS
LIN {X -108.7565,Y -21.7892,Z 110,A -172.2759,B 24.9436,C -1.7348,E1 24.8432,E2 258.0776} C_DIS
LIN {X -107.9171,Y -25.6286,Z 110,A -170.3705,B 24.9443,C -1.7236,E1 24.8444,E2 256.1876} C_DIS
LIN {X -107.1654,Y -28.6033,Z 110,A -168.7748,B 24.9446,C -1.7192,E1 24.8455,E2 254.5933} C_DIS
LIN {X -106.5296,Y -30.893,Z 110,A -167.4085,B 24.9446,C -1.7208,E1 24.8466,E2 253.2153} C_DIS
LIN {X -105.6328,Y -33.8272,Z 110,A -165.8679,B 24.9449,C -1.7143,E1 24.8478,E2 251.6812} C_DIS
LIN {X -104.4347,Y -37.3673,Z 110,A -163.8703,B 24.9451,C -1.7111,E1 24.8497,E2 249.6799} C_DIS
LIN {X -103.4862,Y -39.919,Z 110,A -162.455,B 24.9454,C -1.7073,E1 24.8511,E2 248.2657} C_DIS
LIN {X -102.4754,Y -42.4467,Z 110,A -161.019,B 24.9456,C -1.7044,E1 24.8526,E2 246.8287} C_DIS
LIN {X -101.4028,Y -44.9488,Z 110,A -159.7551,B 24.9462,C -1.6948,E1 24.854,E2 245.5807} C_DIS
LIN {X -100.2692,Y -47.4238,Z 110,A -158.2098,B 24.9461,C -1.6962,E1 24.8559,E2 244.0236} C_DIS
LIN {X -98.8745,Y -50.2629,Z 110,A -156.729,B 24.9467,C -1.6857,E1 24.8577,E2 242.5599} C_DIS
LIN {X -97.6565,Y -52.5908,Z 110,A -155.4946,B 24.9473,C -1.6772,E1 24.8593,E2 241.3393} C_DIS
LIN {X -96.5088,Y -54.6716,Z 110,A -154.0962,B 24.9471,C -1.6805,E1 24.8612,E2 239.9257} C_DIS
LIN {X -95.138,Y -57.0235,Z 110,A -152.6817,B 24.9473,C -1.677,E1 24.8632,E2 238.5121} C_DIS
LIN {X -93.5231,Y -59.6323,Z 110,A -151.0879,B 24.9475,C -1.6733,E1 24.8656,E2 236.9191} C_DIS
LIN {X -92.2254,Y -61.6231,Z 110,A -149.8534,B 24.9477,C -1.6703,E1 24.8675,E2 235.6854} C_DIS
LIN {X -90.4844,Y -64.1494,Z 110,A -148.2597,B 24.9479,C -1.6667,E1 24.87,E2 234.0925} C_DIS
LIN {X -88.9125,Y -66.3112,Z 110,A -147.0117,B 24.9485,C -1.658,E1 24.8721,E2 232.8591} C_DIS
LIN {X -87.2278,Y -68.512,Z 110,A -145.4322,B 24.9483,C -1.6604,E1 24.8748,E2 231.2665} C_DIS
LIN {X -85.5035,Y -70.6521,Z 110,A -144.1811,B 24.949,C -1.6504,E1 24.877,E2 230.0334} C_DIS
LIN {X -83.761,Y -72.7096,Z 110,A -142.6055,B 24.9487,C -1.6544,E1 24.8799,E2 228.4411} C_DIS
LIN {X -81.9513,Y -74.7433,Z 110,A -141.3557,B 24.9493,C -1.645,E1 24.8822,E2 227.2081} C_DIS
LIN {X -79.9432,Y -76.8867,Z 110,A -139.7388,B 24.9493,C -1.6456,E1 24.8853,E2 225.5826} C_DIS
LIN {X -77.4629,Y -79.3878,Z 110,A -137.7098,B 24.949,C -1.6501,E1 24.8893,E2 223.5345} C_DIS
LIN {X -75.4913,Y -81.265,Z 110,A -136.4274,B 24.9495,C -1.6422,E1 24.8919,E2 222.2655} C_DIS
LIN {X -73.4742,Y -83.0931,Z 110,A -134.8849,B 24.9493,C -1.6449,E1 24.8952,E2 220.7106} C_DIS
LIN {X -71.1468,Y -85.0924,Z 110,A -133.5867,B 24.9502,C -1.6304,E1 24.8979,E2 219.4419} C_DIS
LIN {X -69.3085,Y -86.5983,Z 110,A -132.0609,B 24.9496,C -1.64,E1 24.9012,E2 217.8874} C_DIS
LIN {X -66.8858,Y -88.4809,Z 110,A -130.763,B 24.9505,C -1.6257,E1 24.904,E2 216.6189} C_DIS
LIN {X -64.9759,Y -89.8948,Z 110,A -129.2378,B 24.9499,C -1.6355,E1 24.9075,E2 215.0649} C_DIS
LIN {X -62.4637,Y -91.6562,Z 110,A -127.9402,B 24.9507,C -1.6213,E1 24.9105,E2 213.7967} C_DIS
LIN {X -60.4867,Y -92.9747,Z 110,A -126.4153,B 24.9501,C -1.6314,E1 24.9141,E2 212.2429} C_DIS
LIN {X -57.8911,Y -94.6108,Z 110,A -124.9555,B 24.9506,C -1.6239,E1 24.9175,E2 210.7962} C_DIS
LIN {X -55.5518,Y -96.003,Z 110,A -123.5446,B 24.9506,C -1.6221,E1 24.9209,E2 209.3854} C_DIS
LIN {X -53.1623,Y -97.3465,Z 110,A -122.0701,B 24.9506,C -1.6225,E1 24.9245,E2 207.9056} C_DIS
LIN {X -49.8702,Y -99.0752,Z 110,A -120.0683,B 24.9506,C -1.6234,E1 24.9295,E2 205.8964} C_DIS
LIN {X -47.1102,Y -100.4152,Z 110,A -118.6092,B 24.951,C -1.6163,E1 24.9332,E2 204.4503} C_DIS
LIN {X -44.9488,Y -101.4028,Z 110,A -117.2488,B 24.9508,C -1.6204,E1 24.9367,E2 203.077} C_DIS
LIN {X -42.4467,Y -102.4754,Z 110,A -115.8079,B 24.9508,C -1.6204,E1 24.9404,E2 201.6329} C_DIS
LIN {X -39.919,Y -103.4862,Z 110,A -114.4304,B 24.951,C -1.6178,E1 24.944,E2 200.2584} C_DIS
LIN {X -36.083,Y -104.8854,Z 110,A -112.4466,B 24.9514,C -1.6108,E1 24.9491,E2 198.2874} C_DIS
LIN {X -33.4981,Y -105.7393,Z 110,A -110.9082,B 24.9511,C -1.6152,E1 24.9533,E2 196.7358} C_DIS
LIN {X -30.893,Y -106.5296,Z 110,A -109.6297,B 24.9515,C -1.6089,E1 24.9567,E2 195.4701} C_DIS
LIN {X -27.7119,Y -107.3989,Z 110,A -107.8973,B 24.9515,C -1.6091,E1 24.9613,E2 193.7346} C_DIS
LIN {X -25.2916,Y -107.995,Z 110,A -106.6487,B 24.9516,C -1.6068,E1 24.9647,E2 192.4899} C_DIS
LIN {X -22.6336,Y -108.5831,Z 110,A -105.3896,B 24.952,C -1.6,E1 24.9681,E2 191.2453} C_DIS
LIN {X -19.962,Y -109.1059,Z 110,A -103.9823,B 24.952,C -1.5995,E1 24.972,E2 189.8376} C_DIS
LIN {X -17.6203,Y -109.5101,Z 110,A -102.4616,B 24.9513,C -1.6114,E1 24.9763,E2 188.2873} C_DIS
LIN {X -14.9275,Y -109.9095,Z 110,A -101.055,B 24.9513,C -1.6111,E1 24.9801,E2 186.8803} C_DIS
LIN {X -12.2257,Y -110.2427,Z 110,A -99.7779,B 24.9517,C -1.6055,E1 24.9837,E2 185.6157} C_DIS
LIN {X -9.5165,Y -110.5096,Z 110,A -98.2417,B 24.9514,C -1.6109,E1 24.988,E2 184.066} C_DIS
LIN {X -6.8016,Y -110.7098,Z 110,A -96.8356,B 24.9514,C -1.6109,E1 24.9919,E2 182.6593} C_DIS
LIN {X -4.0826,Y -110.8434,Z 110,A -95.4297,B 24.9514,C -1.611,E1 24.9958,E2 181.2528} C_DIS
LIN {X -1.3611,Y -110.9102,Z 110,A -94.0238,B 24.9514,C -1.6112,E1 24.9997,E2 179.8463} C_DIS
LIN {X -1.3611,Y -110.9102,Z 110,A -94.0238,B 24.9514,C -1.6112,E1 24.9997,E2 179.8463} C_DIS
Enddeposition()
LIN {X 0.763,Y -109.9667,Z 110,A -93.2513,B 24.9512,C -1.6142,E1 25.0019,E2 179.0668} C_DIS
Startdeposition()
$VEL.CP = VEL_PRINT
LIN {X -1.4273,Y -109.9648,Z 110,A -94.8322,B 24.9523,C -1.5955,E1 24.9974,E2 180.692} C_DIS
LIN {X -4.5442,Y -109.8786,Z 110,A -96.5998,B 24.9527,C -1.5894,E1 24.9924,E2 182.4744} C_DIS
LIN {X -8.2701,Y -109.6621,Z 110,A -98.525,B 24.9527,C -1.5902,E1 24.987,E2 184.3985} C_DIS
LIN {X -11.4948,Y -109.37,Z 110,A -100.2202,B 24.9527,C -1.59,E1 24.9823,E2 186.095} C_DIS
LIN {X -15.4235,Y -108.8855,Z 110,A -102.2065,B 24.9524,C -1.5935,E1 24.9768,E2 188.0744} C_DIS
LIN {X -18.8089,Y -108.354,Z 110,A -103.97,B 24.9524,C -1.5949,E1 24.972,E2 189.8363} C_DIS
LIN {X -21.8877,Y -107.7725,Z 110,A -105.8406,B 24.9529,C -1.5858,E1 24.9668,E2 191.7305} C_DIS
LIN {X -25.4588,Y -106.9868,Z 110,A -107.6859,B 24.9527,C -1.5892,E1 24.9618,E2 193.5702} C_DIS
LIN {X -28.9018,Y -106.1069,Z 110,A -109.4215,B 24.9523,C -1.595,E1 24.9571,E2 195.2945} C_DIS
LIN {X -32.4475,Y -105.0767,Z 110,A -111.6126,B 24.9529,C -1.5856,E1 24.9512,E2 197.5117} C_DIS
LIN {X -36.4946,Y -103.7404,Z 110,A -113.6044,B 24.9522,C -1.5967,E1 24.946,E2 199.4811} C_DIS
LIN {X -39.6969,Y -102.5592,Z 110,A -115.5795,B 24.9526,C -1.5904,E1 24.9408,E2 201.4752} C_DIS
LIN {X -44.1734,Y -100.711,Z 110,A -117.7566,B 24.9516,C -1.6069,E1 24.9353,E2 203.6179} C_DIS
LIN {X -46.8892,Y -99.4767,Z 110,A -119.4384,B 24.9518,C -1.6036,E1 24.931,E2 205.3119} C_DIS
LIN {X -49.9687,Y -97.9646,Z 110,A -121.4798,B 24.9523,C -1.5957,E1 24.9258,E2 207.3774} C_DIS
LIN {X -52.9636,Y -96.3802,Z 110,A -123.5252,B 24.9528,C -1.587,E1 24.9208,E2 209.4494} C_DIS
LIN {X -56.148,Y -94.5589,Z 110,A -125.5182,B 24.9528,C -1.5866,E1 24.916,E2 211.4494} C_DIS
LIN {X -59.6112,Y -92.4148,Z 110,A -126.9762,B 24.9511,C -1.616,E1 24.9127,E2 212.842} C_DIS
LIN {X -62.2678,Y -90.6478,Z 110,A -128.6372,B 24.9509,C -1.6187,E1 24.9088,E2 214.5022} C_DIS
LIN {X -64.7993,Y -88.854,Z 110,A -130.3819,B 24.951,C -1.6165,E1 24.9048,E2 216.2584} C_DIS
LIN {X -67.7216,Y -86.6491,Z 110,A -132.4874,B 24.9513,C -1.6121,E1 24.9001,E2 218.3819} C_DIS
LIN {X -71.1206,Y -83.88,Z 110,A -134.5641,B 24.9505,C -1.6246,E1 24.8957,E2 220.4369} C_DIS
LIN {X -73.6868,Y -81.6357,Z 110,A -136.4009,B 24.9505,C -1.6257,E1 24.8919,E2 222.2783} C_DIS
LIN {X -76.0014,Y -79.4853,Z 110,A -138.0847,B 24.9504,C -1.6276,E1 24.8885,E2 223.9644} C_DIS
LIN {X -78.5611,Y -76.9564,Z 110,A -139.9986,B 24.9502,C -1.6301,E1 24.8847,E2 225.8805} C_DIS
LIN {X -81.0471,Y -74.3324,Z 110,A -141.9226,B 24.95,C -1.6327,E1 24.881,E2 227.8067} C_DIS
LIN {X -83.5418,Y -71.5176,Z 110,A -143.826,B 24.9496,C -1.6394,E1 24.8776,E2 229.7029} C_DIS
LIN {X -86.1095,Y -68.4043,Z 110,A -145.953,B 24.9494,C -1.6435,E1 24.8738,E2 231.8301} C_DIS
LIN {X -88.617,Y -65.1229,Z 110,A -148.0299,B 24.9489,C -1.6516,E1 24.8703,E2 233.8976} C_DIS
LIN {X -90.6838,Y -62.2161,Z 110,A -150.0705,B 24.949,C -1.6493,E1 24.8671,E2 235.9537} C_DIS
LIN {X -92.5898,Y -59.3386,Z 110,A -151.6888,B 24.9483,C -1.6609,E1 24.8646,E2 237.5525} C_DIS
LIN {X -94.4504,Y -56.3316,Z 110,A -153.3725,B 24.9476,C -1.6718,E1 24.8622,E2 239.2189} C_DIS
LIN {X -95.5254,Y -54.4881,Z 110,A -154.7593,B 24.9481,C -1.6643,E1 24.8602,E2 240.6308} C_DIS
LIN {X -97.2586,Y -51.3294,Z 110,A -156.5546,B 24.9476,C -1.6726,E1 24.8579,E2 242.4158} C_DIS
LIN {X -98.7983,Y -48.3031,Z 110,A -158.6102,B 24.9479,C -1.6666,E1 24.8553,E2 244.4967} C_DIS
LIN {X -100.8518,Y -43.8503,Z 110,A -160.8904,B 24.9468,C -1.6844,E1 24.8527,E2 246.7471} C_DIS
LIN {X -102.2662,Y -40.4429,Z 110,A -162.6831,B 24.9462,C -1.6949,E1 24.8508,E2 248.5248} C_DIS
LIN {X -103.1597,Y -38.108,Z 110,A -164.2535,B 24.9466,C -1.6886,E1 24.8493,E2 250.119} C_DIS
LIN {X -104.444,Y -34.4345,Z 110,A -166.0944,B 24.9457,C -1.7017,E1 24.8476,E2 251.9392} C_DIS
LIN {X -105.2783,Y -31.7915,Z 110,A -167.8101,B 24.9461,C -1.6958,E1 24.8462,E2 253.6787} C_DIS
LIN {X -106.2116,Y -28.5141,Z 110,A -169.3952,B 24.9453,C -1.7084,E1 24.845,E2 255.243} C_DIS
LIN {X -106.9835,Y -25.4725,Z 110,A -171.2092,B 24.9454,C -1.7067,E1 24.8438,E2 257.0717} C_DIS
LIN {X -107.7577,Y -21.96,Z 110,A -173.5282,B 24.9461,C -1.696,E1 24.8425,E2 259.43} C_DIS
LIN {X -108.4771,Y -18.0736,Z 110,A -175.036,B 24.9444,C -1.7231,E1 24.8418,E2 260.8821} C_DIS
LIN {X -109.2859,Y -12.2798,Z 110,A -178.0409,B 24.9436,C -1.7343,E1 24.8407,E2 263.8781} C_DIS
LIN {X -109.5756,Y -9.3525,Z 110,A -179.7226,B 24.9436,C -1.7336,E1 24.8403,E2 265.5716} C_DIS
LIN {X -109.8324,Y -5.5707,Z 110,A 178.2098,B 24.9435,C -1.7365,E1 24.8399,E2 267.6447} C_DIS
LIN {X -109.9667,Y -1.2808,Z 110,A 176.238,B 24.9424,C -1.7537,E1 24.8398,E2 269.5875} C_DIS
LIN {X -109.9685,Y 1.0217,Z 110,A 174.7731,B 24.9428,C -1.7476,E1 24.8398,E2 271.0756} C_DIS
LIN {X -109.803,Y 6.1027,Z 110,A 172.6291,B 24.9409,C -1.7752,E1 24.84,E2 273.1669} C_DIS
LIN {X -109.6455,Y 8.4783,Z 110,A 170.6957,B 24.9424,C -1.7532,E1 24.8404,E2 275.1643} C_DIS
LIN {X -109.1818,Y 13.1687,Z 110,A 168.4288,B 24.9414,C -1.7682,E1 24.8411,E2 277.4091} C_DIS
LIN {X -108.6733,Y 16.8535,Z 110,A 166.536,B 24.9409,C -1.7761,E1 24.8419,E2 279.2941} C_DIS
LIN {X -108.1532,Y 19.9259,Z 110,A 164.6498,B 24.9412,C -1.7715,E1 24.8428,E2 281.2025} C_DIS
LIN {X -107.1357,Y 24.817,Z 110,A 162.2817,B 24.94,C -1.7887,E1 24.8442,E2 283.5437} C_DIS
LIN {X -105.9418,Y 29.5046,Z 110,A 159.5079,B 24.9401,C -1.7872,E1 24.8462,E2 286.3371} C_DIS
LIN {X -104.8263,Y 33.2532,Z 110,A 157.7945,B 24.9389,C -1.8057,E1 24.8476,E2 288.0162} C_DIS
LIN {X -103.5032,Y 37.1663,Z 110,A 155.5129,B 24.9388,C -1.8076,E1 24.8497,E2 290.3062} C_DIS
LIN {X -101.4125,Y 42.5378,Z 110,A 152.8185,B 24.9373,C -1.8285,E1 24.8524,E2 292.9659} C_DIS
LIN {X -98.805,Y 48.2895,Z 110,A 149.1368,B 24.9377,C -1.8236,E1 24.8567,E2 296.6794} C_DIS
LIN {X -97.2902,Y 51.2693,Z 110,A 147.4271,B 24.9372,C -1.83,E1 24.8589,E2 298.383} C_DIS
LIN {X -95.849,Y 53.9167,Z 110,A 145.9742,B 24.9366,C -1.839,E1 24.8609,E2 299.8221} C_DIS
LIN {X -94.2176,Y 56.7203,Z 110,A 144.3395,B 24.9361,C -1.846,E1 24.8632,E2 301.4486} C_DIS
LIN {X -92.3261,Y 59.7494,Z 110,A 142.3195,B 24.9361,C -1.8453,E1 24.8662,E2 303.4806} C_DIS
LIN {X -90.2007,Y 62.911,Z 110,A 140.2763,B 24.9359,C -1.8486,E1 24.8694,E2 305.526} C_DIS
LIN {X -88.4554,Y 65.3436,Z 110,A 138.5871,B 24.9359,C -1.848,E1 24.8722,E2 307.2249} C_DIS
LIN {X -82.9668,Y 72.1836,Z 110,A 134.4259,B 24.9341,C -1.8755,E1 24.8795,E2 311.3399} C_DIS
LIN {X -80.5284,Y 74.896,Z 110,A 132.0294,B 24.9351,C -1.8614,E1 24.884,E2 313.7806} C_DIS
LIN {X -78.5336,Y 76.9843,Z 110,A 129.7906,B 24.9367,C -1.8373,E1 24.8886,E2 316.0862} C_DIS
LIN {X -74.6046,Y 80.7973,Z 110,A 128.0705,B 24.9332,C -1.887,E1 24.8918,E2 317.6951} C_DIS
LIN {X -70.1396,Y 84.7018,Z 110,A 124.0045,B 24.9354,C -1.8568,E1 24.9007,E2 321.8489} C_DIS
LIN {X -66.4224,Y 87.6482,Z 110,A 122.4238,B 24.9326,C -1.896,E1 24.904,E2 323.3419} C_DIS
LIN {X -63.5721,Y 89.7366,Z 110,A 120.1174,B 24.9336,C -1.8819,E1 24.9093,E2 325.69} C_DIS
LIN {X -58.7231,Y 92.9829,Z 110,A 117.4764,B 24.9321,C -1.9032,E1 24.9153,E2 328.289} C_DIS
LIN {X -55.7657,Y 94.7849,Z 110,A 115.5889,B 24.9321,C -1.9032,E1 24.9199,E2 330.182} C_DIS
LIN {X -52.7256,Y 96.5093,Z 110,A 113.5572,B 24.9324,C -1.8983,E1 24.9249,E2 332.2314} C_DIS
LIN {X -49.2503,Y 98.3278,Z 110,A 111.0666,B 24.9334,C -1.8844,E1 24.9312,E2 334.7619} C_DIS
LIN {X -45.501,Y 100.1185,Z 110,A 109.51,B 24.9315,C -1.9113,E1 24.935,E2 336.2584} C_DIS
LIN {X -42.5328,Y 101.4146,Z 110,A 107.8056,B 24.9314,C -1.9131,E1 24.9393,E2 337.9624} C_DIS
LIN {X -38.942,Y 102.8467,Z 110,A 105.4084,B 24.9323,C -1.9008,E1 24.9457,E2 340.3938} C_DIS
LIN {X -35.8487,Y 103.9671,Z 110,A 103.9416,B 24.9314,C -1.9126,E1 24.9495,E2 341.8355} C_DIS
LIN {X -32.147,Y 105.1699,Z 110,A 101.5851,B 24.9322,C -1.902,E1 24.9558,E2 344.2212} C_DIS
LIN {X -28.8472,Y 106.1216,Z 110,A 100.3684,B 24.9304,C -1.9265,E1 24.959,E2 345.3817} C_DIS
LIN {X -26.1403,Y 106.8205,Z 110,A 98.8229,B 24.9306,C -1.9244,E1 24.9632,E2 346.9344} C_DIS
LIN {X -23.3426,Y 107.4666,Z 110,A 97.3043,B 24.9306,C -1.9248,E1 24.9673,E2 348.4539} C_DIS
LIN {X -20.1207,Y 108.1181,Z 110,A 95.1462,B 24.9317,C -1.9085,E1 24.9733,E2 350.6531} C_DIS
LIN {X -16.9351,Y 108.6607,Z 110,A 93.8797,B 24.9304,C -1.9263,E1 24.9767,E2 351.8786} C_DIS
LIN {X -13.7052,Y 109.1159,Z 110,A 92.0949,B 24.9306,C -1.9239,E1 24.9817,E2 353.6703} C_DIS
LIN {X -10.4224,Y 109.4779,Z 110,A 90.4977,B 24.9302,C -1.9298,E1 24.9861,E2 355.2545} C_DIS
LIN {X -6.9798,Y 109.7516,Z 110,A 88.7859,B 24.9299,C -1.9341,E1 24.9908,E2 356.9568} C_DIS
LIN {X -4.3268,Y 109.888,Z 110,A 87.3054,B 24.9301,C -1.9307,E1 24.995,E2 358.4457} C_DIS
LIN {X -1.337,Y 109.9663,Z 110,A 85.7626,B 24.9301,C -1.9317,E1 24.9993,E2 359.9863} C_DIS
LIN {X 2.2095,Y 109.9504,Z 110,A 83.8217,B 24.9303,C -1.9282,E1 25.0047,E2 361.9352} C_DIS
LIN {X 6.0926,Y 109.8035,Z 110,A 81.8972,B 24.93,C -1.9324,E1 25.01,E2 363.8491} C_DIS
LIN {X 9.3071,Y 109.5792,Z 110,A 80.1348,B 24.9302,C -1.9289,E1 25.015,E2 365.619} C_DIS
LIN {X 12.8792,Y 109.2157,Z 110,A 78.2494,B 24.9303,C -1.928,E1 25.0202,E2 367.5052} C_DIS
LIN {X 16.9879,Y 108.6526,Z 110,A 76.0324,B 24.9305,C -1.9251,E1 25.0264,E2 369.7271} C_DIS
LIN {X 21.5718,Y 107.8374,Z 110,A 73.821,B 24.93,C -1.9329,E1 25.0324,E2 371.9175} C_DIS
LIN {X 24.1361,Y 107.293,Z 110,A 72.2586,B 24.9306,C -1.9241,E1 25.0367,E2 373.4987} C_DIS
LIN {X 27.463,Y 106.4881,Z 110,A 70.5604,B 24.9304,C -1.9266,E1 25.0413,E2 375.1884} C_DIS
LIN {X 32.0321,Y 105.2055,Z 110,A 68.2036,B 24.9302,C -1.9296,E1 25.0476,E2 377.5341} C_DIS
LIN {X 35.8345,Y 103.9721,Z 110,A 65.7053,B 24.9316,C -1.9106,E1 25.0543,E2 380.0726} C_DIS
LIN {X 39.4694,Y 102.647,Z 110,A 63.8293,B 24.9313,C -1.9145,E1 25.0591,E2 381.9354} C_DIS
LIN {X 42.3505,Y 101.4915,Z 110,A 62.312,B 24.9311,C -1.917,E1 25.063,E2 383.4434} C_DIS
LIN {X 45.5503,Y 100.0963,Z 110,A 60.5026,B 24.9312,C -1.9153,E1 25.0676,E2 385.2523} C_DIS
LIN {X 49.2482,Y 98.3298,Z 110,A 58.5027,B 24.931,C -1.9183,E1 25.0726,E2 387.2396} C_DIS
LIN {X 52.2942,Y 96.7434,Z 110,A 55.8016,B 24.9339,C -1.8777,E1 25.0795,E2 390.0291} C_DIS
LIN {X 56.8347,Y 94.148,Z 110,A 54.1653,B 24.9309,C -1.9195,E1 25.0832,E2 391.5617} C_DIS
LIN {X 59.4385,Y 92.5257,Z 110,A 52.331,B 24.9318,C -1.9069,E1 25.0876,E2 393.4197} C_DIS
LIN {X 62.4642,Y 90.5113,Z 110,A 50.3573,B 24.9323,C -1.9004,E1 25.0922,E2 395.4022} C_DIS
LIN {X 65.8016,Y 88.1146,Z 110,A 48.3118,B 24.9323,C -1.9007,E1 25.0968,E2 397.4397} C_DIS
LIN {X 69.0705,Y 85.576,Z 110,A 46.0691,B 24.9328,C -1.8931,E1 25.1017,E2 399.6922} C_DIS
LIN {X 71.6592,Y 83.4212,Z 110,A 44.3353,B 24.933,C -1.8905,E1 25.1054,E2 401.4252} C_DIS
LIN {X 74.1808,Y 81.1862,Z 110,A 42.6068,B 24.9332,C -1.8882,E1 25.109,E2 403.1524} C_DIS
LIN {X 76.4188,Y 79.0829,Z 110,A 41.0868,B 24.9332,C -1.8882,E1 25.112,E2 404.6659} C_DIS
LIN {X 79.2778,Y 76.2166,Z 110,A 39.0387,B 24.9332,C -1.8863,E1 25.116,E2 406.7098} C_DIS
LIN {X 81.5889,Y 73.7391,Z 110,A 37.1819,B 24.9339,C -1.8784,E1 25.1195,E2 408.5771} C_DIS
LIN {X 83.7999,Y 71.2147,Z 110,A 35.546,B 24.9338,C -1.8792,E1 25.1225,E2 410.2038} C_DIS
LIN {X 85.9433,Y 68.6147,Z 110,A 33.8716,B 24.9338,C -1.8785,E1 25.1255,E2 411.872} C_DIS
LIN {X 87.2802,Y 66.9043,Z 110,A 32.6607,B 24.9343,C -1.8723,E1 25.1275,E2 413.0918} C_DIS
LIN {X 89.4143,Y 64.0239,Z 110,A 30.6828,B 24.9349,C -1.8629,E1 25.1308,E2 415.0825} C_DIS
LIN {X 91.6571,Y 60.77,Z 110,A 28.6081,B 24.9354,C -1.8569,E1 25.1341,E2 417.161} C_DIS
LIN {X 93.8087,Y 57.3931,Z 110,A 26.5919,B 24.9355,C -1.8544,E1 25.1371,E2 419.1728} C_DIS
LIN {X 95.4555,Y 54.6097,Z 110,A 24.6461,B 24.9366,C -1.8385,E1 25.1398,E2 421.1462} C_DIS
LIN {X 97.3559,Y 51.1445,Z 110,A 22.9276,B 24.936,C -1.8477,E1 25.142,E2 422.8339} C_DIS
LIN {X 99.9622,Y 45.8462,Z 110,A 19.9742,B 24.9362,C -1.8444,E1 25.1456,E2 425.7793} C_DIS
LIN {X 101.5946,Y 42.1057,Z 110,A 17.8135,B 24.9368,C -1.8367,E1 25.148,E2 427.9464} C_DIS
LIN {X 102.4811,Y 39.8958,Z 110,A 16.4018,B 24.9375,C -1.8255,E1 25.1495,E2 429.3765} C_DIS
LIN {X 103.7893,Y 36.3554,Z 110,A 14.5491,B 24.9375,C -1.8247,E1 25.1512,E2 431.2208} C_DIS
LIN {X 105.4535,Y 31.2009,Z 110,A 12.0235,B 24.9373,C -1.8292,E1 25.1533,E2 433.7213} C_DIS
LIN {X 106.3859,Y 27.8607,Z 110,A 9.7773,B 24.939,C -1.8042,E1 25.155,E2 436.0137} C_DIS
LIN {X 107.4189,Y 23.5614,Z 110,A 7.6713,B 24.9389,C -1.8058,E1 25.1563,E2 438.1037} C_DIS
LIN {X 108.2277,Y 19.5115,Z 110,A 5.8901,B 24.9382,C -1.8155,E1 25.1573,E2 439.8516} C_DIS
LIN {X 108.5354,Y 17.7249,Z 110,A 4.5018,B 24.9398,C -1.7928,E1 25.1579,E2 441.2854} C_DIS
LIN {X 109.0672,Y 14.0814,Z 110,A 2.6646,B 24.9399,C -1.7903,E1 25.1586,E2 443.1176} C_DIS
LIN {X 109.4193,Y 11.0239,Z 110,A 1.0085,B 24.9404,C -1.7828,E1 25.1591,E2 444.7816} C_DIS
LIN {X 109.7626,Y 6.8089,Z 110,A -1.1867,B 24.9409,C -1.776,E1 25.1596,E2 446.9796} C_DIS
LIN {X 109.9172,Y 3.4859,Z 110,A -2.7597,B 24.9408,C -1.7776,E1 25.1597,E2 448.5397} C_DIS
LIN {X 109.9737,Y 0.2771,Z 110,A -4.6161,B 24.9417,C -1.7639,E1 25.1597,E2 450.4172} C_DIS
LIN {X 109.9253,Y -3.2227,Z 110,A -6.3395,B 24.9417,C -1.7625,E1 25.1597,E2 452.1337} C_DIS
LIN {X 109.7867,Y -6.3972,Z 110,A -8.0476,B 24.9423,C -1.7548,E1 25.1594,E2 453.8499} C_DIS
LIN {X 109.496,Y -10.2261,Z 110,A -9.956,B 24.9424,C -1.7524,E1 25.159,E2 455.7527} C_DIS
LIN {X 109.1636,Y -13.3237,Z 110,A -11.6392,B 24.943,C -1.7444,E1 25.1584,E2 457.4447} C_DIS
LIN {X 108.6965,Y -16.7038,Z 110,A -13.3411,B 24.9431,C -1.742,E1 25.1577,E2 459.1421} C_DIS
LIN {X 108.1079,Y -20.1745,Z 110,A -15.0252,B 24.9431,C -1.7428,E1 25.1569,E2 460.8147} C_DIS
LIN {X 107.5495,Y -22.9624,Z 110,A -16.6711,B 24.9439,C -1.7307,E1 25.156,E2 462.4795} C_DIS
LIN {X 106.7549,Y -26.4092,Z 110,A -18.3314,B 24.9437,C -1.7329,E1 25.1549,E2 464.1249} C_DIS
LIN {X 106.0034,Y -29.2847,Z 110,A -19.885,B 24.9441,C -1.7277,E1 25.1538,E2 465.6819} C_DIS
LIN {X 105.0896,Y -32.4058,Z 110,A -21.331,B 24.9437,C -1.7334,E1 25.1527,E2 467.106} C_DIS
LIN {X 104.0943,Y -35.4745,Z 110,A -23.0392,B 24.9441,C -1.7269,E1 25.1512,E2 468.82} C_DIS
LIN {X 102.6984,Y -39.3338,Z 110,A -25.5617,B 24.9456,C -1.7031,E1 25.1487,E2 471.3846} C_DIS
LIN {X 101.2116,Y -43.0146,Z 110,A -27.4135,B 24.9454,C -1.7063,E1 25.1468,E2 473.2185} C_DIS
LIN {X 99.9288,Y -45.9181,Z 110,A -29.2703,B 24.9463,C -1.6923,E1 25.1446,E2 475.0984} C_DIS
LIN {X 98.6869,Y -48.5278,Z 110,A -30.6563,B 24.9463,C -1.693,E1 25.1429,E2 476.4751} C_DIS
LIN {X 97.071,Y -51.6855,Z 110,A -32.6824,B 24.9471,C -1.6796,E1 25.1403,E2 478.5221} C_DIS
LIN {X 94.8108,Y -55.7217,Z 110,A -35.1949,B 24.9479,C -1.6681,E1 25.1367,E2 481.0489} C_DIS
LIN {X 92.2001,Y -59.9456,Z 110,A -37.355,B 24.9471,C -1.6795,E1 25.1336,E2 483.1711} C_DIS
LIN {X 90.4627,Y -62.5342,Z 110,A -38.8814,B 24.9471,C -1.6793,E1 25.1312,E2 484.6905} C_DIS
LIN {X 88.7649,Y -64.9209,Z 110,A -40.509,B 24.9477,C -1.6706,E1 25.1285,E2 486.3308} C_DIS
LIN {X 86.7331,Y -67.6142,Z 110,A -42.2373,B 24.9479,C -1.6671,E1 25.1256,E2 488.0591} C_DIS
LIN {X 84.1811,Y -70.7661,Z 110,A -44.436,B 24.9485,C -1.6577,E1 25.1217,E2 490.2698} C_DIS
LIN {X 82.101,Y -73.167,Z 110,A -46.0867,B 24.9488,C -1.6536,E1 25.1186,E2 491.9227} C_DIS
LIN {X 80.0466,Y -75.4088,Z 110,A -47.6291,B 24.9488,C -1.6515,E1 25.1157,E2 493.4635} C_DIS
LIN {X 77.5024,Y -78.0218,Z 110,A -49.5928,B 24.9494,C -1.644,E1 25.1118,E2 495.4365} C_DIS
LIN {X 75.0532,Y -80.381,Z 110,A -51.1113,B 24.9489,C -1.6508,E1 25.1088,E2 496.9325} C_DIS
LIN {X 73.1754,Y -82.0935,Z 110,A -52.5186,B 24.9493,C -1.6441,E1 25.1059,E2 498.35} C_DIS
LIN {X 70.6533,Y -84.2749,Z 110,A -54.4022,B 24.95,C -1.6337,E1 25.1018,E2 500.2509} C_DIS
LIN {X 68.1928,Y -86.2767,Z 110,A -55.9353,B 24.9499,C -1.6353,E1 25.0985,E2 501.7745} C_DIS
LIN {X 65.5057,Y -88.3366,Z 110,A -57.6452,B 24.9499,C -1.6338,E1 25.0947,E2 503.4816} C_DIS
LIN {X 62.1801,Y -90.7077,Z 110,A -59.9762,B 24.9508,C -1.6207,E1 25.0893,E2 505.8357} C_DIS
LIN {X 59.1052,Y -92.7396,Z 110,A -61.7267,B 24.9506,C -1.6243,E1 25.0852,E2 507.5719} C_DIS
LIN {X 54.9908,Y -95.2365,Z 110,A -63.9782,B 24.9502,C -1.6307,E1 25.0799,E2 509.8012} C_DIS
LIN {X 52.5311,Y -96.6148,Z 110,A -66.6295,B 24.9534,C -1.5774,E1 25.0731,E2 512.571} C_DIS
LIN {X 47.6515,Y -99.1124,Z 110,A -68.574,B 24.9513,C -1.6116,E1 25.0685,E2 514.4295} C_DIS
LIN {X 44.2172,Y -100.6919,Z 110,A -70.2804,B 24.9508,C -1.6198,E1 25.0642,E2 516.1121} C_DIS
LIN {X 40.4117,Y -102.2784,Z 110,A -72.6684,B 24.9516,C -1.6064,E1 25.0579,E2 518.5262} C_DIS
LIN {X 37.1016,Y -103.5267,Z 110,A -74.6309,B 24.9521,C -1.5988,E1 25.0528,E2 520.5026} C_DIS
LIN {X 33.2462,Y -104.8286,Z 110,A -76.939,B 24.9527,C -1.5882,E1 25.0466,E2 522.8314} C_DIS
LIN {X 29.7902,Y -105.8608,Z 110,A -78.8651,B 24.953,C -1.5842,E1 25.0414,E2 524.7638} C_DIS
LIN {X 26.6776,Y -106.6882,Z 110,A -80.4931,B 24.953,C -1.5846,E1 25.037,E2 526.3885} C_DIS
LIN {X 23.0615,Y -107.5279,Z 110,A -82.205,B 24.9525,C -1.5922,E1 25.0324,E2 528.0802} C_DIS
LIN {X 19.0612,Y -108.3087,Z 110,A -84.1484,B 24.9522,C -1.598,E1 25.0271,E2 530.0076} C_DIS
LIN {X 15.9457,Y -108.8113,Z 110,A -86.101,B 24.953,C -1.5839,E1 25.0216,E2 531.9918} C_DIS
LIN {X 10.9883,Y -109.4231,Z 110,A -88.5849,B 24.9528,C -1.5873,E1 25.0147,E2 534.4659} C_DIS
LIN {X 6.7807,Y -109.765,Z 110,A -90.5892,B 24.9524,C -1.5944,E1 25.0092,E2 536.4524} C_DIS
LIN {X 3.5676,Y -109.9147,Z 110,A -92.3273,B 24.9526,C -1.5912,E1 25.0043,E2 538.1975} C_DIS
LIN {X 0.763,Y -109.9667,Z 110,A -93.2493,B 24.9512,C -1.6134,E1 25.0019,E2 539.0668} C_DIS
Enddeposition()
LIN {X 0.763,Y -109.9667,Z 110,A -93.2493,B 24.9512,C -1.6134,E1 25.0019,E2 539.0668} C_DIS
Startdeposition()
$VEL.CP = VEL_PRINT
LIN {X 3.1015,Y -108.9845,Z 110,A -91.8447,B 24.9498,C -1.6374,E1 25.006,E2 537.6054} C_DIS
LIN {X 6.3387,Y -108.8444,Z 110,A -90.0936,B 24.9496,C -1.6401,E1 25.0109,E2 535.8485} C_DIS
LIN {X 9.6971,Y -108.5967,Z 110,A -88.3546,B 24.9496,C -1.6397,E1 25.0157,E2 534.1114} C_DIS
LIN {X 13.39,Y -108.2048,Z 110,A -85.6868,B 24.9477,C -1.6713,E1 25.0233,E2 531.3709} C_DIS
LIN {X 17.8865,Y -107.5512,Z 110,A -84.021,B 24.9495,C -1.6423,E1 25.0277,E2 529.7753} C_DIS
LIN {X 21.487,Y -106.891,Z 110,A -82.0345,B 24.9492,C -1.6466,E1 25.0332,E2 527.781} C_DIS
LIN {X 25.1375,Y -106.0927,Z 110,A -79.8882,B 24.9486,C -1.6563,E1 25.0391,E2 525.6148} C_DIS
LIN {X 32.6604,Y -104.0222,Z 110,A -75.9335,B 24.9487,C -1.6546,E1 25.0497,E2 521.6708} C_DIS
LIN {X 36.935,Y -102.5826,Z 110,A -73.694,B 24.9489,C -1.652,E1 25.0556,E2 519.4419} C_DIS
LIN {X 39.9151,Y -101.4592,Z 110,A -72.0302,B 24.9487,C -1.6539,E1 25.0599,E2 517.7772} C_DIS
LIN {X 43.0396,Y -100.1754,Z 110,A -70.3569,B 24.9489,C -1.6521,E1 25.0642,E2 516.1121} C_DIS
LIN {X 47.4641,Y -98.155,Z 110,A -68.1269,B 24.9495,C -1.642,E1 25.0698,E2 513.9114} C_DIS
LIN {X 49.9654,Y -96.9061,Z 110,A -65.624,B 24.9465,C -1.6893,E1 25.0763,E2 511.3036} C_DIS
LIN {X 53.6961,Y -94.8909,Z 110,A -63.9319,B 24.9477,C -1.6698,E1 25.0803,E2 509.6625} C_DIS
LIN {X 58.6767,Y -91.8928,Z 110,A -60.8737,B 24.9474,C -1.6758,E1 25.0875,E2 506.6} C_DIS
LIN {X 62.0321,Y -89.6619,Z 110,A -58.8446,B 24.9474,C -1.6762,E1 25.0922,E2 504.5768} C_DIS
LIN {X 64.1075,Y -88.1904,Z 110,A -57.0203,B 24.9458,C -1.7004,E1 25.0964,E2 502.7018} C_DIS
LIN {X 67.1409,Y -85.904,Z 110,A -55.2895,B 24.9463,C -1.693,E1 25.1002,E2 500.9948} C_DIS
LIN {X 70.542,Y -83.1327,Z 110,A -53.1929,B 24.9465,C -1.689,E1 25.1047,E2 498.9156} C_DIS
LIN {X 73.8686,Y -80.1913,Z 110,A -50.6351,B 24.9456,C -1.7044,E1 25.11,E2 496.3319} C_DIS
LIN {X 78.1725,Y -76.003,Z 110,A -47.6814,B 24.9456,C -1.7031,E1 25.1158,E2 493.3936} C_DIS
LIN {X 80.9001,Y -73.0931,Z 110,A -45.6653,B 24.9456,C -1.7049,E1 25.1196,E2 491.3821} C_DIS
LIN {X 84.1489,Y -69.3279,Z 110,A -42.9462,B 24.9448,C -1.7164,E1 25.1246,E2 488.6483} C_DIS
LIN {X 87.6167,Y -64.8911,Z 110,A -40.0558,B 24.9445,C -1.7214,E1 25.1295,E2 485.7599} C_DIS
LIN {X 89.9493,Y -61.617,Z 110,A -37.6689,B 24.9433,C -1.7395,E1 25.1333,E2 483.3419} C_DIS
LIN {X 93.6133,Y -55.8925,Z 110,A -34.2387,B 24.943,C -1.7434,E1 25.1383,E2 479.9198} C_DIS
LIN {X 95.2838,Y -52.9926,Z 110,A -32.0791,B 24.9415,C -1.7666,E1 25.1413,E2 477.7168} C_DIS
LIN {X 97.4252,Y -48.9474,Z 110,A -30.4816,B 24.9434,C -1.7376,E1 25.1433,E2 476.1963} C_DIS
LIN {X 99.4375,Y -44.7142,Z 110,A -27.9157,B 24.9426,C -1.7496,E1 25.1463,E2 473.6158} C_DIS
LIN {X 100.9439,Y -41.201,Z 110,A -25.8683,B 24.9421,C -1.7575,E1 25.1485,E2 471.561} C_DIS
LIN {X 102.488,Y -37.1942,Z 110,A -23.0671,B 24.94,C -1.789,E1 25.1513,E2 468.7012} C_DIS
LIN {X 103.8715,Y -33.1375,Z 110,A -21.3705,B 24.9412,C -1.7711,E1 25.1527,E2 467.0565} C_DIS
LIN {X 105.2061,Y -28.6163,Z 110,A -18.9061,B 24.9407,C -1.7784,E1 25.1546,E2 464.589} C_DIS
LIN {X 106.1576,Y -24.8567,Z 110,A -16.9532,B 24.9405,C -1.7811,E1 25.1559,E2 462.641} C_DIS
LIN {X 106.9067,Y -21.4104,Z 110,A -14.7616,B 24.9391,C -1.8023,E1 25.1571,E2 460.4123} C_DIS
LIN {X 107.847,Y -16.019,Z 110,A -12.3288,B 24.9398,C -1.7917,E1 25.1582,E2 458.0188} C_DIS
LIN {X 108.2696,Y -12.8409,Z 110,A -10.6045,B 24.9393,C -1.7989,E1 25.1588,E2 456.2876} C_DIS
LIN {X 108.6198,Y -9.4477,Z 110,A -8.8027,B 24.9389,C -1.8051,E1 25.1593,E2 454.4818} C_DIS
LIN {X 108.8475,Y -6.2833,Z 110,A -7.1396,B 24.9386,C -1.8104,E1 25.1596,E2 452.8162} C_DIS
LIN {X 109.0034,Y -2.3593,Z 110,A -5.082,B 24.9381,C -1.8168,E1 25.1598,E2 450.7557} C_DIS
LIN {X 109.0235,Y 1.1425,Z 110,A -3.2482,B 24.9377,C -1.8225,E1 25.1598,E2 448.9195} C_DIS
LIN {X 108.957,Y 3.9984,Z 110,A -1.6649,B 24.9372,C -1.831,E1 25.1596,E2 447.3255} C_DIS
LIN {X 108.747,Y 7.8423,Z 110,A 0.2693,B 24.937,C -1.8336,E1 25.1593,E2 445.3967} C_DIS
LIN {X 108.4309,Y 11.3983,Z 110,A 2.0486,B 24.9369,C -1.8353,E1 25.1588,E2 443.6239} C_DIS
LIN {X 108.0054,Y 14.9064,Z 110,A 4.0962,B 24.9359,C -1.8497,E1 25.158,E2 441.5544} C_DIS
LIN {X 107.3495,Y 19.0609,Z 110,A 6.8562,B 24.9336,C -1.8814,E1 25.1567,E2 438.7359} C_DIS
LIN {X 106.4129,Y 23.7431,Z 110,A 8.6422,B 24.9354,C -1.8567,E1 25.1557,E2 437.0184} C_DIS
LIN {X 105.741,Y 26.5775,Z 110,A 10.8399,B 24.9329,C -1.8913,E1 25.1541,E2 434.7517} C_DIS
LIN {X 104.5438,Y 30.9481,Z 110,A 12.863,B 24.9336,C -1.8825,E1 25.1526,E2 432.7609} C_DIS
LIN {X 103.5799,Y 34.0388,Z 110,A 14.2824,B 24.9341,C -1.8751,E1 25.1514,E2 431.3671} C_DIS
LIN {X 102.4791,Y 37.2189,Z 110,A 15.9667,B 24.934,C -1.8766,E1 25.1498,E2 429.6887} C_DIS
LIN {X 101.1484,Y 40.6987,Z 110,A 17.9506,B 24.9335,C -1.8835,E1 25.1477,E2 427.6995} C_DIS
LIN {X 100.1191,Y 43.1687,Z 110,A 19.3459,B 24.9332,C -1.8871,E1 25.1462,E2 426.3034} C_DIS
LIN {X 99.0808,Y 45.5027,Z 110,A 21.3753,B 24.9308,C -1.9215,E1 25.1438,E2 424.2039} C_DIS
LIN {X 97.0128,Y 49.7566,Z 110,A 23.0729,B 24.9328,C -1.8934,E1 25.1417,E2 422.5814} C_DIS
LIN {X 95.7893,Y 52.0731,Z 110,A 24.7673,B 24.9315,C -1.9113,E1 25.1394,E2 420.8539} C_DIS
LIN {X 93.3751,Y 56.2887,Z 110,A 27.0487,B 24.9319,C -1.9061,E1 25.1362,E2 418.5963} C_DIS
LIN {X 91.966,Y 58.5627,Z 110,A 28.5009,B 24.9315,C -1.9119,E1 25.134,E2 417.138} C_DIS
LIN {X 89.962,Y 61.5982,Z 110,A 30.2422,B 24.9317,C -1.9093,E1 25.1313,E2 415.4113} C_DIS
LIN {X 87.4354,Y 65.1339,Z 110,A 32.6143,B 24.931,C -1.9189,E1 25.1274,E2 413.028} C_DIS
LIN {X 85.2124,Y 68.0169,Z 110,A 34.5334,B 24.9306,C -1.9238,E1 25.1241,E2 411.1065} C_DIS
LIN {X 82.9529,Y 70.7531,Z 110,A 36.3291,B 24.9306,C -1.9252,E1 25.1209,E2 409.3156} C_DIS
LIN {X 80.785,Y 73.2213,Z 110,A 38.1889,B 24.9298,C -1.9349,E1 25.1174,E2 407.4412} C_DIS
LIN {X 77.5722,Y 76.6142,Z 110,A 40.49,B 24.9299,C -1.9336,E1 25.113,E2 405.153} C_DIS
LIN {X 74.9215,Y 79.2089,Z 110,A 42.3165,B 24.9299,C -1.9324,E1 25.1093,E2 403.337} C_DIS
LIN {X 72.8621,Y 81.1069,Z 110,A 43.7471,B 24.9299,C -1.9336,E1 25.1064,E2 401.9093} C_DIS
LIN {X 70.4555,Y 83.2064,Z 110,A 45.6854,B 24.9289,C -1.9481,E1 25.1022,E2 399.9444} C_DIS
LIN {X 67.2889,Y 85.7878,Z 110,A 47.6336,B 24.9292,C -1.9435,E1 25.098,E2 398.0142} C_DIS
LIN {X 63.8316,Y 88.3917,Z 110,A 50.1169,B 24.9282,C -1.9565,E1 25.0924,E2 395.5092} C_DIS
LIN {X 60.7394,Y 90.5435,Z 110,A 51.9914,B 24.9283,C -1.9553,E1 25.0881,E2 393.6439} C_DIS
LIN {X 57.3145,Y 92.7497,Z 110,A 54.1433,B 24.928,C -1.9591,E1 25.083,E2 391.49} C_DIS
LIN {X 51.3857,Y 96.1597,Z 110,A 57.8299,B 24.9274,C -1.9681,E1 25.074,E2 387.793} C_DIS
LIN {X 48.4223,Y 97.6855,Z 110,A 59.6145,B 24.9271,C -1.9717,E1 25.0696,E2 386.0047} C_DIS
LIN {X 44.1893,Y 99.6741,Z 110,A 62.1252,B 24.9267,C -1.9767,E1 25.0632,E2 383.4882} C_DIS
LIN {X 40.5402,Y 101.2129,Z 110,A 63.8642,B 24.9276,C -1.9645,E1 25.0587,E2 381.7822} C_DIS
LIN {X 37.5294,Y 102.3658,Z 110,A 65.7024,B 24.9271,C -1.9722,E1 25.0539,E2 379.9298} C_DIS
LIN {X 33.7028,Y 103.6886,Z 110,A 67.7773,B 24.9271,C -1.9718,E1 25.0484,E2 377.8599} C_DIS
LIN {X 30.5441,Y 104.6636,Z 110,A 69.6482,B 24.9266,C -1.9786,E1 25.0434,E2 375.976} C_DIS
LIN {X 23.8143,Y 106.3974,Z 110,A 73.0638,B 24.9272,C -1.9709,E1 25.0342,E2 372.5837} C_DIS
LIN {X 18.2792,Y 107.4855,Z 110,A 76.1576,B 24.9267,C -1.9774,E1 25.0257,E2 369.478} C_DIS
LIN {X 13.6715,Y 108.1683,Z 110,A 78.5298,B 24.9269,C -1.9749,E1 25.0191,E2 367.1138} C_DIS
LIN {X 10.283,Y 108.5427,Z 110,A 80.3082,B 24.9269,C -1.9746,E1 25.0142,E2 365.3372} C_DIS
LIN {X 6.7107,Y 108.823,Z 110,A 82.4193,B 24.9262,C -1.984,E1 25.0083,E2 363.2049} C_DIS
LIN {X 2.5964,Y 108.999,Z 110,A 84.4348,B 24.9267,C -1.9777,E1 25.0027,E2 361.2047} C_DIS
LIN {X -0.7077,Y 109.026,Z 110,A 86.1049,B 24.9269,C -1.9747,E1 24.998,E2 359.5418} C_DIS
LIN {X -3.5522,Y 108.9707,Z 110,A 87.9237,B 24.9259,C -1.9874,E1 24.9929,E2 357.6926} C_DIS
LIN {X -7.1579,Y 108.7933,Z 110,A 89.7025,B 24.9264,C -1.9819,E1 24.9879,E2 355.9264} C_DIS
LIN {X -11.3359,Y 108.4374,Z 110,A 91.7199,B 24.927,C -1.9732,E1 24.9824,E2 353.9284} C_DIS
LIN {X -15.0809,Y 107.9806,Z 110,A 94.0187,B 24.9261,C -1.9848,E1 24.9759,E2 351.6006} C_DIS
LIN {X -20.3182,Y 107.1188,Z 110,A 97.2608,B 24.9249,C -2.0009,E1 24.9669,E2 348.3167} C_DIS
LIN {X -25.042,Y 106.1147,Z 110,A 98.861,B 24.9279,C -1.9609,E1 24.9628,E2 346.8095} C_DIS
LIN {X -32.3187,Y 104.1282,Z 110,A 103.0468,B 24.9276,C -1.9654,E1 24.9515,E2 342.6063} C_DIS
LIN {X -36.5326,Y 102.7266,Z 110,A 105.6115,B 24.9271,C -1.9717,E1 24.9447,E2 340.0219} C_DIS
LIN {X -42.0092,Y 100.6108,Z 110,A 108.4915,B 24.928,C -1.9593,E1 24.9373,E2 337.1649} C_DIS
LIN {X -44.8122,Y 99.3934,Z 110,A 110.0893,B 24.9282,C -1.9566,E1 24.9332,E2 335.5697} C_DIS
LIN {X -49.9444,Y 96.9168,Z 110,A 113.0549,B 24.9287,C -1.9506,E1 24.9258,E2 332.6106} C_DIS
LIN {X -52.861,Y 95.3573,Z 110,A 114.8326,B 24.9287,C -1.9492,E1 24.9214,E2 330.8313} C_DIS
LIN {X -55.4841,Y 93.8546,Z 110,A 116.8034,B 24.9279,C -1.9613,E1 24.9166,E2 328.8259} C_DIS
LIN {X -58.3679,Y 92.091,Z 110,A 118.398,B 24.9287,C -1.9508,E1 24.9129,E2 327.2512} C_DIS
LIN {X -62.1057,Y 89.6107,Z 110,A 120.9939,B 24.9283,C -1.9554,E1 24.9069,E2 324.6355} C_DIS
LIN {X -64.9782,Y 87.5523,Z 110,A 122.3393,B 24.93,C -1.9316,E1 24.904,E2 323.3419} C_DIS
LIN {X -66.6954,Y 86.2493,Z 110,A 124.0383,B 24.9286,C -1.9512,E1 24.9001,E2 321.5901} C_DIS
LIN {X -69.5076,Y 83.9995,Z 110,A 126.1597,B 24.9283,C -1.9559,E1 24.8955,E2 319.4493} C_DIS
LIN {X -72.9258,Y 81.0499,Z 110,A 127.9528,B 24.9303,C -1.928,E1 24.8919,E2 317.7157} C_DIS
LIN {X -78.0919,Y 76.0867,Z 110,A 132.3244,B 24.9293,C -1.9423,E1 24.8831,E2 313.2916} C_DIS
LIN {X -81.1082,Y 72.8607,Z 110,A 134.0796,B 24.9313,C -1.9146,E1 24.8799,E2 311.5945} C_DIS
LIN {X -83.2298,Y 70.4281,Z 110,A 136.5016,B 24.9296,C -1.9381,E1 24.8755,E2 309.1054} C_DIS
LIN {X -86.3903,Y 66.5124,Z 110,A 138.3565,B 24.9323,C -1.9007,E1 24.8724,E2 307.3308} C_DIS
LIN {X -89.2871,Y 62.5713,Z 110,A 140.7287,B 24.9333,C -1.8861,E1 24.8685,E2 304.9819} C_DIS
LIN {X -92.1101,Y 58.3382,Z 110,A 143.5418,B 24.9335,C -1.8838,E1 24.8642,E2 302.1602} C_DIS
LIN {X -94.7782,Y 53.8935,Z 110,A 146.3623,B 24.9338,C -1.8796,E1 24.8602,E2 299.3352} C_DIS
LIN {X -96.3848,Y 50.9625,Z 110,A 148.0891,B 24.9342,C -1.8733,E1 24.8579,E2 297.6143} C_DIS
LIN {X -98.0819,Y 47.6164,Z 110,A 150.5758,B 24.9333,C -1.8869,E1 24.8548,E2 295.0816} C_DIS
LIN {X -99.5939,Y 44.3672,Z 110,A 152.2081,B 24.9343,C -1.8717,E1 24.853,E2 293.4767} C_DIS
Enddeposition()
END
